METHOD PROTECTED M_ProcessFCR : BOOL
(**************************************************************************************
 * 	Application		:	BoxControl Framework
 *	Revision		:	$Revision: 404529 $
 *	Revision date	:	$Date: 2018-04-23 08:21:38 +0200 (Mo., 23 Apr 2018) $
 *	Last changed by	:	$Author: b7bolm $
 *	URL				:	$URL: http://almscdc.swisslog.com/repo/SWPD/Development/BoxControlFramework/20_Release/trunk/01_Software/BCF/BCF/JumpStart/20_Product/10_App/11_Com/10_Lib/10_Conv/12_MFCS/11_SIS/FB_SIS_MsgManager_6_1.TcPOU $
 *
 *	Purpose			:	Send FCR
 *
 * ------------------------------------------------------------------------------------
 *	Copyright Swisslog [IP AG], Switzerland. All rights reserved.
 * 
 * ------------------------------------------------------------------------------------
 *	
 * 	Revision History: 
 *
 * 	VERSION			DATE			INITIALS			DESCRIPTION
 *	0.1				01.01.2001		swl					Example
 *
 **************************************************************************************)
VAR_INPUT
 	meChannelSrc		: E_MFCS_Channel; // Source communicaton channel
	mpFCR				: POINTER TO ST_ITC_FCR; // Pointer to FCR
END_VAR
(**************************************************************************************************************
 	Check if a telegram needs to be send
***************************************************************************************************************)
// If settings allow sending a FCR 	
IF  Settings.Telegrams.SendFCR THEN
	// If the source of the request is this channel or is undefined
	IF meChannelSrc = Settings.MFCS_Channel OR
		meChannelSrc = E_MFCS_Channel.BEGIN_CHANNEL THEN
		;//Proceed
	ELSE // Source is a different MFCS Connection
		// Dont send a telegram		
		RETURN;
	END_IF	
ELSE
	// Dont send a telegram		
	RETURN;
END_IF

(**************************************************************************************************************
 	ITC - Map generic data to type
***************************************************************************************************************)
MEMCPY(destAddr := ADR(FCR_ITC), srcAddr := mpFCR, n := SIZEOF(FCR_ITC));

(**************************************************************************************************************
 	Formatting data
***************************************************************************************************************)

// Fill position
FCR.Position	:= 	F_StuffString(
						InputString 	:= FCR_ITC.Position, 
						StringLength	:= SIS_6_1.POSITION_STRINGLENGTH, 
						StuffCharacter 	:= '0',
						LeftAligned		:= FALSE);

// Fill code
FCR.Code	:= F_StuffString(
				InputString 	:= INT_TO_STRING(FCR_ITC.Code), 
				StringLength	:= SIS_6_1.CONTROLCODE_STRINGLENGTH, 
				StuffCharacter 	:= '0',
				LeftAligned		:= FALSE);

// Fill variable
FCR.Variable 	:= F_StuffString(
					InputString 	:= DINT_TO_STRING(FCR_ITC.Variable), 
					StringLength	:= SIS_6_1.CONTROLVARIABLE_STRINGLENGTH, 
					StuffCharacter 	:= '0',
					LeftAligned		:= FALSE);

// Fill errorcode
FCR.ReturnCode 	:= F_StuffString(
					InputString 	:= INT_TO_STRING(FCR_ITC.ReturnCode), 
					StringLength	:= SIS_6_1.ERRORCODE_STRINGLENGTH, 
					StuffCharacter 	:= '0',
					LeftAligned		:= FALSE);


(**************************************************************************************************************
 	Build string and add to Base Driver
***************************************************************************************************************)
MEMSET(destAddr := ADR(SendTelegram), 0, SIZEOF(SendTelegram));
WritePointer := 0;

F_AssembleByteStream(
	pSrc:= ADR('FCR'), 
	SrcLen:= 3, 
	pDest:= ADR(SendTelegram), 
	DestLen:= SIZEOF(SendTelegram), 
	WritePointer:= WritePointer);

F_AssembleByteStream(
	pSrc:= ADR(FCR.Position), 
	SrcLen:= INT_TO_UDINT(LEN(FCR.Position)), 
	pDest:= ADR(SendTelegram), 
	DestLen:= SIZEOF(SendTelegram), 
	WritePointer:= WritePointer);	
	
F_AssembleByteStream(
	pSrc:= ADR(FCR.Code), 
	SrcLen:= INT_TO_UDINT(LEN(FCR.Code)), 
	pDest:= ADR(SendTelegram), 
	DestLen:= SIZEOF(SendTelegram), 
	WritePointer:= WritePointer);	
	
F_AssembleByteStream(
	pSrc:= ADR(FCR.Variable), 
	SrcLen:= INT_TO_UDINT(LEN(FCR.Variable)), 
	pDest:= ADR(SendTelegram), 
	DestLen:= SIZEOF(SendTelegram), 
	WritePointer:= WritePointer);	
	
F_AssembleByteStream(
	pSrc:= ADR(FCR.ReturnCode), 
	SrcLen:= INT_TO_UDINT(LEN(FCR.ReturnCode)), 
	pDest:= ADR(SendTelegram), 
	DestLen:= SIZEOF(SendTelegram), 
	WritePointer:= WritePointer);	

// Add to buffer of Base Driver
M_ProcessFCR := fbBaseDriver.M_SendAppData(
					mpSendData := ADR(SendTelegram),
					mSendDataLen := WritePointer);
					
// Forward to mirror channel
M_MirrorData(Data := ADR(SendTelegram), DataLen := WritePointer);
END_METHOD

METHOD PROTECTED M_ProcessFSR : BOOL
(**************************************************************************************
 * 	Application		:	BoxControl Framework
 *	Revision		:	$Revision: 404529 $
 *	Revision date	:	$Date: 2018-04-23 08:21:38 +0200 (Mo., 23 Apr 2018) $
 *	Last changed by	:	$Author: b7bolm $
 *	URL				:	$URL: http://almscdc.swisslog.com/repo/SWPD/Development/BoxControlFramework/20_Release/trunk/01_Software/BCF/BCF/JumpStart/20_Product/10_App/11_Com/10_Lib/10_Conv/12_MFCS/11_SIS/FB_SIS_MsgManager_6_1.TcPOU $
 *
 *	Purpose			:	Send FSR
 *
 * ------------------------------------------------------------------------------------
 *	Copyright Swisslog [IP AG], Switzerland. All rights reserved.
 * 
 * ------------------------------------------------------------------------------------
 *	
 * 	Revision History: 
 *
 * 	VERSION			DATE			INITIALS			DESCRIPTION
 *	0.1				01.01.2001		swl					Example
 *
 **************************************************************************************)
VAR_INPUT
 	meChannelSrc		: E_MFCS_Channel; // Source communicaton channel
	mpFSR				: POINTER TO ST_ITC_FSR; // Pointer to FSR
END_VAR
(**************************************************************************************************************
 	Check if a telegram needs to be send
***************************************************************************************************************)
// If settings allow sending a FSR 	
IF  Settings.Telegrams.SendFSR THEN
	// If the source of the request is this channel or is undefined
	IF meChannelSrc = Settings.MFCS_Channel OR
		meChannelSrc = E_MFCS_Channel.BEGIN_CHANNEL THEN
		;//Proceed
	ELSE // Source is a different MFCS Connection
		// Dont send a telegram		
		RETURN;
	END_IF	
ELSE
	// Dont send a telegram		
	RETURN;
END_IF

(**************************************************************************************************************
 	ITC - Map generic data to type
***************************************************************************************************************)
MEMCPY(destAddr := ADR(FSR_ITC), srcAddr := mpFSR, n := SIZEOF(FSR_ITC));

(**************************************************************************************************************
 	Formatting data
***************************************************************************************************************)
// Set position
FSR.Position := F_StuffString(
					InputString 	:= FSR_ITC.Position, 
					StringLength	:= SIS_6_1.POSITION_STRINGLENGTH, 
					StuffCharacter 	:= '0',
					LeftAligned		:= FALSE);
					
// Set previous function no
FSR.PrevFunctionNo := F_StuffString(
						InputString 	:= FSR_ITC.PrevFunctionNo, 
						StringLength	:= SIS_6_1.POSITION_STRINGLENGTH, 
						StuffCharacter 	:= '0',
						LeftAligned		:= FALSE);
						
// Set next function no
FSR.NextFunctionNo := F_StuffString(
						InputString 	:= FSR_ITC.NextFunctionNo, 
						StringLength	:= SIS_6_1.POSITION_STRINGLENGTH, 
						StuffCharacter 	:= '0',
						LeftAligned		:= FALSE);
						
// Set state
FSR.State := INT_TO_STRING(FSR_ITC.eState);

// Set enabled
FSR.Enabled := INT_TO_STRING(BOOL_TO_INT(FSR_ITC.Enabled));

//modifications needed BCFD-10111FSR data incorrect (M_ProcessFSR)
// Set transport state
FSR.TransportState := F_StuffString(
						InputString 	:= INT_TO_STRING(TO_INT(FSR_ITC.TransportState)), 
						StringLength	:= SIS_6_1.FSR_STATES_STRINGLENGTH, 
						StuffCharacter 	:= '0',
						LeftAligned		:= FALSE);

// Set takeover state	
FSR.TakeOverState := F_StuffString(
						InputString 	:= INT_TO_STRING(TO_INT(FSR_ITC.TakeOverState)), 
						StringLength	:= SIS_6_1.FSR_STATES_STRINGLENGTH, 
						StuffCharacter 	:= '0',
						LeftAligned		:= FALSE);

// Set handover state
FSR.HandOverState := F_StuffString(
						InputString 	:= INT_TO_STRING(TO_INT(FSR_ITC.HandOverState)), 
						StringLength	:= SIS_6_1.FSR_STATES_STRINGLENGTH, 
						StuffCharacter 	:= '0',
						LeftAligned		:= FALSE);

// Set TU-ID
FSR.TU_ID := F_StuffString(
				InputString 	:= FSR_ITC.TU_ID, 
				StringLength	:= SIS_6_1.TU_ID_STRINGLENGTH, 
				StuffCharacter 	:= ' ',
				LeftAligned		:= FALSE);

// Set TU-Type	
FSR.TU_Type := F_StuffString(
				InputString 	:= INT_TO_STRING(FSR_ITC.TU_Type), 
				StringLength	:= SIS_6_1.TU_TYPE_STRINGLENGTH, 
				StuffCharacter 	:= '0',
				LeftAligned		:= FALSE);
				
// Set Assignment ID	
FSR.AssignmentID := F_StuffString(
						InputString 	:= UDINT_TO_STRING(FSR_ITC.AssignmentID), 
						StringLength	:= SIS_6_1.ASSIGNMENT_ID_STRINGLENGTH, 
						StuffCharacter 	:= '0',
						LeftAligned		:= FALSE);

// Set load information	
FSR.LoadInformation  := INT_TO_STRING(FSR_ITC.LoadInformation);

// Set destination
FSR.Destination  := F_StuffString(
						InputString 	:= FSR_ITC.Destination, 
						StringLength	:= SIS_6_1.POSITION_STRINGLENGTH, 
						StuffCharacter 	:= '0',
						LeftAligned		:= FALSE);
						
// Set error state
FSR.ErrorState := INT_TO_STRING(FSR_ITC.eErrorState);

// Set error code				
FSR.ErrorCode := F_StuffString(
					InputString 	:= INT_TO_STRING(FSR_ITC.eErrorCode), 
					StringLength	:= SIS_6_1.ERRORCODE_STRINGLENGTH, 
					StuffCharacter 	:= '0',
					LeftAligned		:= FALSE);
					
// Set error type		
FSR.ErrorType  := INT_TO_STRING(FSR_ITC.eErrorType);

// Set error information	
FSR.ErrorInformation  := F_StuffString(
							InputString 	:= FSR_ITC.ErrorInformation, 
							StringLength	:= SIS_6_1.ERRORINFORMATION_STRINGLENGTH, 
							StuffCharacter 	:= ' ',
							LeftAligned		:= TRUE);
// Set variable		
FSR.Variable := F_StuffString(
					InputString 	:= DINT_TO_STRING(FSR_ITC.Variable), 
					StringLength	:= SIS_6_1.FSR_VARIABLE_STRINGLENGTH, 
					StuffCharacter 	:= '0',
					LeftAligned		:= FALSE);

// Get Error Code 
FSR.ReturnCode := F_StuffString(
					InputString 	:= INT_TO_STRING(FSR_ITC.eReturnCode), 
					StringLength	:= SIS_6_1.ERRORCODE_STRINGLENGTH, 
					StuffCharacter 	:= '0',
					LeftAligned		:= FALSE);
					
(**************************************************************************************************************
 	Build string and add to Base Driver
***************************************************************************************************************)
MEMSET(destAddr := ADR(SendTelegram), 0, SIZEOF(SendTelegram));
WritePointer := 0;

F_AssembleByteStream(
	pSrc:= ADR('FSR'), 
	SrcLen:= 3, 
	pDest:= ADR(SendTelegram), 
	DestLen:= SIZEOF(SendTelegram), 
	WritePointer:= WritePointer);

F_AssembleByteStream(
	pSrc:= ADR(FSR.Position), 
	SrcLen:= INT_TO_UDINT(LEN(FSR.Position)), 
	pDest:= ADR(SendTelegram), 
	DestLen:= SIZEOF(SendTelegram), 
	WritePointer:= WritePointer);	

F_AssembleByteStream(
	pSrc:= ADR(FSR.PrevFunctionNo), 
	SrcLen:= INT_TO_UDINT(LEN(FSR.PrevFunctionNo)), 
	pDest:= ADR(SendTelegram), 
	DestLen:= SIZEOF(SendTelegram), 
	WritePointer:= WritePointer);	

F_AssembleByteStream(
	pSrc:= ADR(FSR.NextFunctionNo), 
	SrcLen:= INT_TO_UDINT(LEN(FSR.NextFunctionNo)), 
	pDest:= ADR(SendTelegram), 
	DestLen:= SIZEOF(SendTelegram), 
	WritePointer:= WritePointer);	
	
F_AssembleByteStream(
	pSrc:= ADR(FSR.State), 
	SrcLen:= INT_TO_UDINT(LEN(FSR.State)), 
	pDest:= ADR(SendTelegram), 
	DestLen:= SIZEOF(SendTelegram), 
	WritePointer:= WritePointer);	
	
F_AssembleByteStream(
	pSrc:= ADR(FSR.Enabled), 
	SrcLen:= INT_TO_UDINT(LEN(FSR.Enabled)), 
	pDest:= ADR(SendTelegram), 
	DestLen:= SIZEOF(SendTelegram), 
	WritePointer:= WritePointer);	
	
F_AssembleByteStream(
	pSrc:= ADR(FSR.TransportState), 
	SrcLen:= INT_TO_UDINT(LEN(FSR.TransportState)), 
	pDest:= ADR(SendTelegram), 
	DestLen:= SIZEOF(SendTelegram), 
	WritePointer:= WritePointer);	
	
F_AssembleByteStream(
	pSrc:= ADR(FSR.TakeOverState), 
	SrcLen:= INT_TO_UDINT(LEN(FSR.TakeOverState)), 
	pDest:= ADR(SendTelegram), 
	DestLen:= SIZEOF(SendTelegram), 
	WritePointer:= WritePointer);	
	
F_AssembleByteStream(
	pSrc:= ADR(FSR.HandOverState), 
	SrcLen:= INT_TO_UDINT(LEN(FSR.HandOverState)), 
	pDest:= ADR(SendTelegram), 
	DestLen:= SIZEOF(SendTelegram), 
	WritePointer:= WritePointer);	

F_AssembleByteStream(
	pSrc:= ADR(FSR.TU_ID), 
	SrcLen:= INT_TO_UDINT(LEN(FSR.TU_ID)), 
	pDest:= ADR(SendTelegram), 
	DestLen:= SIZEOF(SendTelegram), 
	WritePointer:= WritePointer);	
	
F_AssembleByteStream(
	pSrc:= ADR(FSR.TU_Type), 
	SrcLen:= INT_TO_UDINT(LEN(FSR.TU_Type)), 
	pDest:= ADR(SendTelegram), 
	DestLen:= SIZEOF(SendTelegram), 
	WritePointer:= WritePointer);	

F_AssembleByteStream(
	pSrc:= ADR(FSR.AssignmentID), 
	SrcLen:= INT_TO_UDINT(LEN(FSR.AssignmentID)), 
	pDest:= ADR(SendTelegram), 
	DestLen:= SIZEOF(SendTelegram), 
	WritePointer:= WritePointer);	

F_AssembleByteStream(
	pSrc:= ADR(FSR.LoadInformation), 
	SrcLen:= INT_TO_UDINT(LEN(FSR.LoadInformation)), 
	pDest:= ADR(SendTelegram), 
	DestLen:= SIZEOF(SendTelegram), 
	WritePointer:= WritePointer);	
	
F_AssembleByteStream(
	pSrc:= ADR(FSR.Destination), 
	SrcLen:= INT_TO_UDINT(LEN(FSR.Destination)), 
	pDest:= ADR(SendTelegram), 
	DestLen:= SIZEOF(SendTelegram), 
	WritePointer:= WritePointer);	

F_AssembleByteStream(
	pSrc:= ADR(FSR.ErrorState), 
	SrcLen:= INT_TO_UDINT(LEN(FSR.ErrorState)), 
	pDest:= ADR(SendTelegram), 
	DestLen:= SIZEOF(SendTelegram), 
	WritePointer:= WritePointer);	
		
F_AssembleByteStream(
	pSrc:= ADR(FSR.ErrorCode), 
	SrcLen:= INT_TO_UDINT(LEN(FSR.ErrorCode)), 
	pDest:= ADR(SendTelegram), 
	DestLen:= SIZEOF(SendTelegram), 
	WritePointer:= WritePointer);	
	
F_AssembleByteStream(
	pSrc:= ADR(FSR.ErrorType), 
	SrcLen:= INT_TO_UDINT(LEN(FSR.ErrorType)), 
	pDest:= ADR(SendTelegram), 
	DestLen:= SIZEOF(SendTelegram), 
	WritePointer:= WritePointer);	
	
F_AssembleByteStream(
	pSrc:= ADR(FSR.ErrorInformation), 
	SrcLen:= INT_TO_UDINT(LEN(FSR.ErrorInformation)), 
	pDest:= ADR(SendTelegram), 
	DestLen:= SIZEOF(SendTelegram), 
	WritePointer:= WritePointer);	
	
F_AssembleByteStream(
	pSrc:= ADR(FSR.Variable), 
	SrcLen:= INT_TO_UDINT(LEN(FSR.Variable)), 
	pDest:= ADR(SendTelegram), 
	DestLen:= SIZEOF(SendTelegram), 
	WritePointer:= WritePointer);	
	
F_AssembleByteStream(
	pSrc:= ADR(FSR.ReturnCode), 
	SrcLen:= INT_TO_UDINT(LEN(FSR.ReturnCode)), 
	pDest:= ADR(SendTelegram), 
	DestLen:= SIZEOF(SendTelegram), 
	WritePointer:= WritePointer);	
	

// Add to buffer of Base Driver
M_ProcessFSR := fbBaseDriver.M_SendAppData(
					mpSendData := ADR(SendTelegram),
					mSendDataLen := WritePointer);

// Forward to mirror channel
M_MirrorData(Data := ADR(SendTelegram), DataLen := WritePointer);
END_METHOD

METHOD PROTECTED M_ProcessGCR : BOOL
(**************************************************************************************
 * 	Application		:	BoxControl Framework
 *	Revision		:	$Revision: 404529 $
 *	Revision date	:	$Date: 2018-04-23 08:21:38 +0200 (Mo., 23 Apr 2018) $
 *	Last changed by	:	$Author: b7bolm $
 *	URL				:	$URL: http://almscdc.swisslog.com/repo/SWPD/Development/BoxControlFramework/20_Release/trunk/01_Software/BCF/BCF/JumpStart/20_Product/10_App/11_Com/10_Lib/10_Conv/12_MFCS/11_SIS/FB_SIS_MsgManager_6_1.TcPOU $
 *
 *	Purpose			:	Send GCR
 *
 * ------------------------------------------------------------------------------------
 *	Copyright Swisslog [IP AG], Switzerland. All rights reserved.
 * 
 * ------------------------------------------------------------------------------------
 *	
 * 	Revision History: 
 *
 * 	VERSION			DATE			INITIALS			DESCRIPTION
 *	0.1				01.01.2001		swl					Example
 *
 **************************************************************************************)
VAR_INPUT
 	meChannelSrc		: E_MFCS_Channel; // Source communicaton channel
	mpGCR				: POINTER TO ST_ITC_GCR; // Pointer to GCR
END_VAR
(**************************************************************************************************************
 	Check if a telegram needs to be send
***************************************************************************************************************)
// If settings allow sending a GCR 	
IF  Settings.Telegrams.SendGCR THEN
	// If the source of the request is this channel or is undefined
	IF meChannelSrc = Settings.MFCS_Channel OR
		meChannelSrc = E_MFCS_Channel.BEGIN_CHANNEL THEN
		;//Proceed
	ELSE // Source is a different MFCS Connection
		// Dont send a telegram		
		RETURN;
	END_IF	
ELSE
	// Dont send a telegram		
	RETURN;
END_IF

(**************************************************************************************************************
 	ITC - Map generic data to type
***************************************************************************************************************)
MEMCPY(destAddr := ADR(GCR_ITC), srcAddr := mpGCR, n := SIZEOF(GCR_ITC));

(**************************************************************************************************************
 	Formatting data
***************************************************************************************************************)
// Get SIS-Number 
GCR.GroupName := F_StuffString(
					InputString 	:= GCR_ITC.GroupName, 
					StringLength	:= SIS_6_1.POSITION_STRINGLENGTH, 
					StuffCharacter 	:= '0',
					LeftAligned		:= FALSE);

// Get Code 
GCR.Code := F_StuffString(
				InputString 	:= INT_TO_STRING(GCR_ITC.Code), 
				StringLength	:= SIS_6_1.CONTROLCODE_STRINGLENGTH, 
				StuffCharacter 	:= '0',
				LeftAligned		:= FALSE);

// Get Variable 
GCR.Variable := F_StuffString(
					InputString 	:= DINT_TO_STRING(GCR_ITC.Variable), 
					StringLength	:= SIS_6_1.CONTROLVARIABLE_STRINGLENGTH, 
					StuffCharacter 	:= '0',
					LeftAligned		:= FALSE);

// Get ErrorCode 
GCR.ReturnCode := F_StuffString(
					InputString 	:= INT_TO_STRING(GCR_ITC.ReturnCode), 
					StringLength	:= SIS_6_1.ERRORCODE_STRINGLENGTH, 
					StuffCharacter 	:= '0',
					LeftAligned		:= FALSE);

(**************************************************************************************************************
 	Build string and add to Base Driver
***************************************************************************************************************)
MEMSET(destAddr := ADR(SendTelegram), 0, SIZEOF(SendTelegram));
WritePointer := 0;

F_AssembleByteStream(
	pSrc:= ADR('GCR'), 
	SrcLen:= 3, 
	pDest:= ADR(SendTelegram), 
	DestLen:= SIZEOF(SendTelegram), 
	WritePointer:= WritePointer);

F_AssembleByteStream(
	pSrc:= ADR(GCR.GroupName), 
	SrcLen:= INT_TO_UDINT(LEN(GCR.GroupName)), 
	pDest:= ADR(SendTelegram), 
	DestLen:= SIZEOF(SendTelegram), 
	WritePointer:= WritePointer);	

F_AssembleByteStream(
	pSrc:= ADR(GCR.Code), 
	SrcLen:= INT_TO_UDINT(LEN(GCR.Code)), 
	pDest:= ADR(SendTelegram), 
	DestLen:= SIZEOF(SendTelegram), 
	WritePointer:= WritePointer);	

F_AssembleByteStream(
	pSrc:= ADR(GCR.Variable), 
	SrcLen:= INT_TO_UDINT(LEN(GCR.Variable)), 
	pDest:= ADR(SendTelegram), 
	DestLen:= SIZEOF(SendTelegram), 
	WritePointer:= WritePointer);	

F_AssembleByteStream(
	pSrc:= ADR(GCR.ReturnCode), 
	SrcLen:= INT_TO_UDINT(LEN(GCR.ReturnCode)), 
	pDest:= ADR(SendTelegram), 
	DestLen:= SIZEOF(SendTelegram), 
	WritePointer:= WritePointer);	

// Add to buffer of Base Driver
M_ProcessGCR := fbBaseDriver.M_SendAppData(
					mpSendData := ADR(SendTelegram),
					mSendDataLen := WritePointer);

// Forward to mirror channel
M_MirrorData(Data := ADR(SendTelegram), DataLen := WritePointer);
END_METHOD

METHOD PROTECTED M_ProcessGDR : BOOL
(**************************************************************************************
 * 	Application		:	BoxControl Framework
 *	Revision		:	$Revision: 404529 $
 *	Revision date	:	$Date: 2018-04-23 08:21:38 +0200 (Mo., 23 Apr 2018) $
 *	Last changed by	:	$Author: b7bolm $
 *	URL				:	$URL: http://almscdc.swisslog.com/repo/SWPD/Development/BoxControlFramework/20_Release/trunk/01_Software/BCF/BCF/JumpStart/20_Product/10_App/11_Com/10_Lib/10_Conv/12_MFCS/11_SIS/FB_SIS_MsgManager_6_1.TcPOU $
 *
 *	Purpose			:	Send GDR
 *
 * ------------------------------------------------------------------------------------
 *	Copyright Swisslog [IP AG], Switzerland. All rights reserved.
 * 
 * ------------------------------------------------------------------------------------
 *	
 * 	Revision History: 
 *
 * 	VERSION			DATE			INITIALS			DESCRIPTION
 *	0.1				01.01.2001		swl					Example
 *
 **************************************************************************************)
VAR_INPUT
 	meChannelSrc		: E_MFCS_Channel; // Source communicaton channel
	mpGDR				: POINTER TO ST_ITC_GDR; // Pointer to GDR
END_VAR
(**************************************************************************************************************
 	Check if a telegram needs to be send
***************************************************************************************************************)
// If settings allow sending a GDR 	
IF  Settings.Telegrams.SendGDR THEN
	// If the source of the request is this channel or is undefined
	IF meChannelSrc = Settings.MFCS_Channel OR
		meChannelSrc = E_MFCS_Channel.BEGIN_CHANNEL THEN
		;//Proceed
	ELSE // Source is a different MFCS Connection
		// Dont send a telegram		
		RETURN;
	END_IF	
ELSE
	// Dont send a telegram		
	RETURN;
END_IF

(**************************************************************************************************************
 	ITC - Map generic data to type
***************************************************************************************************************)
MEMCPY(destAddr := ADR(GDR_ITC), srcAddr := mpGDR, n := SIZEOF(GDR_ITC));
MEMSET(destAddr := ADR(GDR), 0, SIZEOF(GDR));
(**************************************************************************************************************
 	Formatting data
***************************************************************************************************************)
// Get SIS-Number 
GDR.Position := F_StuffString(
					InputString 	:= GDR_ITC.Position, 
					StringLength	:= SIS_6_1.POSITION_STRINGLENGTH, 
					StuffCharacter 	:= '0',
					LeftAligned := FALSE);
// Get Variable 
GDR.Variable := F_StuffString(
				InputString 	:= GDR_ITC.Variable, 
				StringLength	:= SIS_6_1.GATHERED_DATA_VARIABLE, 
				StuffCharacter 	:= ' ',
				LeftAligned		:= FALSE);
//Number of Sets
GDR.NumberOfSets := 	F_StuffString(
										InputString 	:=INT_TO_STRING(GDR_ITC.NumberOfSets), 
										StringLength	:= SIS_6_1.DATA_ACQUISITION_NUMBEROFSETS, 
										StuffCharacter 	:= '0',
										LeftAligned		:= FALSE);
//Build Data Set String
FOR Idx:= 0 TO GDR_ITC.NumberOfSets-1 DO 
	GDR.DataSet[Idx]  := CONCAT(GDR.DataSet[Idx],F_StuffString(InputString := GDR_ITC.DataSet[Idx].Value, StringLength:= Conveyor.GATHERED_DATA_VALUE,StuffCharacter := '0', LeftAligned := FALSE));
	GDR.DataSet[Idx]  := CONCAT(GDR.DataSet[Idx],GDR_ITC.DataSet[Idx].TimeStamp);
	GDR.DataSet[Idx]  := CONCAT(GDR.DataSet[Idx],F_StuffString(InputString 	:= INT_TO_STRING(GDR_ITC.DataSet[Idx].Sequence), StringLength:= SIS_6_1.GATHERED_DATA_SEQUENCE,StuffCharacter := '0', LeftAligned := FALSE));
END_FOR;

// Get Error Code 
GDR.ReturnCode := F_StuffString(
				InputString 	:= INT_TO_STRING(GDR_ITC.eReturnCode), 
				StringLength	:= SIS_6_1.ERRORCODE_STRINGLENGTH, 
				StuffCharacter 	:= '0',
				LeftAligned 	:= FALSE);
				
(**************************************************************************************************************
 	Build string and add to Base Driver
***************************************************************************************************************)
MEMSET(destAddr := ADR(SendTelegram), 0, SIZEOF(SendTelegram));
WritePointer := 0;

F_AssembleByteStream(
	pSrc:= ADR('GDR'), 
	SrcLen:= 3, 
	pDest:= ADR(SendTelegram), 
	DestLen:= SIZEOF(SendTelegram), 
	WritePointer:= WritePointer);
	
F_AssembleByteStream(
	pSrc:= ADR(GDR.Position), 
	SrcLen:= INT_TO_UDINT(LEN(GDR.Position)), 
	pDest:= ADR(SendTelegram), 
	DestLen:= SIZEOF(SendTelegram), 
	WritePointer:= WritePointer);

F_AssembleByteStream(
	pSrc:= ADR(GDR.Variable), 
	SrcLen:= INT_TO_UDINT(LEN(GDR.Variable)), 
	pDest:= ADR(SendTelegram), 
	DestLen:= SIZEOF(SendTelegram), 
	WritePointer:= WritePointer);

F_AssembleByteStream(
	pSrc:= ADR(GDR.NumberOfSets), 
	SrcLen:= INT_TO_UDINT(LEN(GDR.NumberOfSets)), 
	pDest:= ADR(SendTelegram), 
	DestLen:= SIZEOF(SendTelegram), 
	WritePointer:= WritePointer);

FOR Idx:= 0
 TO GDR_ITC.NumberOfSets DO
	F_AssembleByteStream(
						pSrc		:= ADR(GDR.DataSet[Idx]), 
						SrcLen		:= INT_TO_UDINT(LEN(GDR.DataSet[Idx])), 
						pDest		:= ADR(SendTelegram),
						DestLen		:= SIZEOF(SendTelegram), 
						WritePointer:= WritePointer);
						
END_FOR

	
	
	
F_AssembleByteStream(
	pSrc:= ADR(GDR.ReturnCode), 
	SrcLen:= INT_TO_UDINT(LEN(GDR.ReturnCode)), 
	pDest:= ADR(SendTelegram), 
	DestLen:= SIZEOF(SendTelegram), 
	WritePointer:= WritePointer);

// Add to buffer of Base Driver
M_ProcessGDR := fbBaseDriver.M_SendAppData(
					mpSendData := ADR(SendTelegram),
					mSendDataLen := WritePointer);

// Forward to mirror channel
M_MirrorData(Data := ADR(SendTelegram), DataLen := WritePointer);
END_METHOD

METHOD PROTECTED M_ProcessGSR : BOOL
(**************************************************************************************
 * 	Application		:	BoxControl Framework
 *	Revision		:	$Revision: 404529 $
 *	Revision date	:	$Date: 2018-04-23 08:21:38 +0200 (Mo., 23 Apr 2018) $
 *	Last changed by	:	$Author: b7bolm $
 *	URL				:	$URL: http://almscdc.swisslog.com/repo/SWPD/Development/BoxControlFramework/20_Release/trunk/01_Software/BCF/BCF/JumpStart/20_Product/10_App/11_Com/10_Lib/10_Conv/12_MFCS/11_SIS/FB_SIS_MsgManager_6_1.TcPOU $
 *
 *	Purpose			:	Send GSR
 *
 * ------------------------------------------------------------------------------------
 *	Copyright Swisslog [IP AG], Switzerland. All rights reserved.
 * 
 * ------------------------------------------------------------------------------------
 *	
 * 	Revision History: 
 *
 * 	VERSION			DATE			INITIALS			DESCRIPTION
 *	0.1				01.01.2001		swl					Example
 *
 **************************************************************************************)
VAR_INPUT
 	meChannelSrc		: E_MFCS_Channel; // Source communicaton channel
	mpGSR				: POINTER TO ST_ITC_GSR; // Pointer to GSR
END_VAR
(**************************************************************************************************************
 	Check if a telegram needs to be send
***************************************************************************************************************)
// If settings allow sending a GSR 	
IF  Settings.Telegrams.SendGSR THEN
	// If the source of the request is this channel or is undefined
	IF meChannelSrc = Settings.MFCS_Channel OR
		meChannelSrc = E_MFCS_Channel.BEGIN_CHANNEL THEN
		;//Proceed
	ELSE // Source is a different MFCS Connection
		// Dont send a telegram		
		RETURN;
	END_IF	
ELSE
	// Dont send a telegram		
	RETURN;
END_IF

(**************************************************************************************************************
 	ITC - Map generic data to type
***************************************************************************************************************)
MEMCPY(destAddr := ADR(GSR_ITC), srcAddr := mpGSR, n := SIZEOF(GSR_ITC));

(**************************************************************************************************************
 	Formatting data
***************************************************************************************************************)
// Get SIS-Number 
GSR.GroupName := F_StuffString(
					InputString 	:= GSR_ITC.GroupName, 
					StringLength	:= SIS_6_1.POSITION_STRINGLENGTH, 
					StuffCharacter 	:= '0',
					LeftAligned		:= FALSE);

// Get Mode 
GSR.Mode := INT_TO_STRING(GSR_ITC.eMode);

// Get State 
GSR.State := INT_TO_STRING(GSR_ITC.eState);

// Get ErrorState 
GSR.ErrorState := INT_TO_STRING(GSR_ITC.eErrorState);

// Get ErrorCode 
GSR.ErrorCode := F_StuffString(
					InputString 	:= INT_TO_STRING(GSR_ITC.eErrorCode), 
					StringLength	:= SIS_6_1.ERRORCODE_STRINGLENGTH, 
					StuffCharacter 	:= '0',
					LeftAligned		:= FALSE);

// Get ErrorType 
GSR.ErrorType := INT_TO_STRING(GSR_ITC.eErrorType);

// Get ErrorInformation 
GSR.ErrorInformation := F_StuffString(
							InputString 	:= GSR_ITC.ErrorInformation, 
							StringLength	:= SIS_6_1.ERRORINFORMATION_STRINGLENGTH, 
							StuffCharacter 	:= ' ',
							LeftAligned		:= TRUE);

// Get Variable 
GSR.Variable := F_StuffString(
					InputString 	:= DINT_TO_STRING(GSR_ITC.Variable), 
					StringLength	:= SIS_6_1.CONTROLVARIABLE_STRINGLENGTH, 
					StuffCharacter 	:= '0',
					LeftAligned		:= FALSE);
					
// Get Error Code 
GSR.ReturnCode := F_StuffString(
					InputString 	:= INT_TO_STRING(GSR_ITC.eReturnCode), 
					StringLength	:= SIS_6_1.ERRORCODE_STRINGLENGTH, 
					StuffCharacter 	:= '0',
					LeftAligned		:= FALSE);

(**************************************************************************************************************
 	Build string and add to Base Driver
***************************************************************************************************************)
MEMSET(destAddr := ADR(SendTelegram), 0, SIZEOF(SendTelegram));
WritePointer := 0;

F_AssembleByteStream(
	pSrc:= ADR('GSR'), 
	SrcLen:= 3, 
	pDest:= ADR(SendTelegram), 
	DestLen:= SIZEOF(SendTelegram), 
	WritePointer:= WritePointer);

F_AssembleByteStream(
	pSrc:= ADR(GSR.GroupName), 
	SrcLen:= INT_TO_UDINT(LEN(GSR.GroupName)), 
	pDest:= ADR(SendTelegram), 
	DestLen:= SIZEOF(SendTelegram), 
	WritePointer:= WritePointer);	
	
F_AssembleByteStream(
	pSrc:= ADR(GSR.Mode), 
	SrcLen:= INT_TO_UDINT(LEN(GSR.Mode)), 
	pDest:= ADR(SendTelegram), 
	DestLen:= SIZEOF(SendTelegram), 
	WritePointer:= WritePointer);	
	
F_AssembleByteStream(
	pSrc:= ADR(GSR.State), 
	SrcLen:= INT_TO_UDINT(LEN(GSR.State)), 
	pDest:= ADR(SendTelegram), 
	DestLen:= SIZEOF(SendTelegram), 
	WritePointer:= WritePointer);	

F_AssembleByteStream(
	pSrc:= ADR(GSR.ErrorState), 
	SrcLen:= INT_TO_UDINT(LEN(GSR.ErrorState)), 
	pDest:= ADR(SendTelegram), 
	DestLen:= SIZEOF(SendTelegram), 
	WritePointer:= WritePointer);	

F_AssembleByteStream(
	pSrc:= ADR(GSR.ErrorCode), 
	SrcLen:= INT_TO_UDINT(LEN(GSR.ErrorCode)), 
	pDest:= ADR(SendTelegram), 
	DestLen:= SIZEOF(SendTelegram), 
	WritePointer:= WritePointer);	
	
F_AssembleByteStream(
	pSrc:= ADR(GSR.ErrorType), 
	SrcLen:= INT_TO_UDINT(LEN(GSR.ErrorType)), 
	pDest:= ADR(SendTelegram), 
	DestLen:= SIZEOF(SendTelegram), 
	WritePointer:= WritePointer);	
	
F_AssembleByteStream(
	pSrc:= ADR(GSR.ErrorInformation), 
	SrcLen:= INT_TO_UDINT(LEN(GSR.ErrorInformation)), 
	pDest:= ADR(SendTelegram), 
	DestLen:= SIZEOF(SendTelegram), 
	WritePointer:= WritePointer);	

F_AssembleByteStream(
	pSrc:= ADR(GSR.Variable), 
	SrcLen:= INT_TO_UDINT(LEN(GSR.Variable)), 
	pDest:= ADR(SendTelegram), 
	DestLen:= SIZEOF(SendTelegram), 
	WritePointer:= WritePointer);	
	
F_AssembleByteStream(
	pSrc:= ADR(GSR.ReturnCode), 
	SrcLen:= INT_TO_UDINT(LEN(GSR.ReturnCode)), 
	pDest:= ADR(SendTelegram), 
	DestLen:= SIZEOF(SendTelegram), 
	WritePointer:= WritePointer);	


// Add to buffer of Base Driver
M_ProcessGSR := fbBaseDriver.M_SendAppData(
					mpSendData := ADR(SendTelegram),
					mSendDataLen := WritePointer);

// Forward to mirror channel
M_MirrorData(Data := ADR(SendTelegram), DataLen := WritePointer);
END_METHOD

METHOD PROTECTED M_ProcessGVR : BOOL
(**************************************************************************************
 * 	Application		:	BoxControl Framework
 *	Revision		:	$Revision: 404529 $
 *	Revision date	:	$Date: 2018-04-23 08:21:38 +0200 (Mo., 23 Apr 2018) $
 *	Last changed by	:	$Author: b7bolm $
 *	URL				:	$URL: http://almscdc.swisslog.com/repo/SWPD/Development/BoxControlFramework/20_Release/trunk/01_Software/BCF/BCF/JumpStart/20_Product/10_App/11_Com/10_Lib/10_Conv/12_MFCS/11_SIS/FB_SIS_MsgManager_6_1.TcPOU $
 *
 *	Purpose			:	Send GVR
 *
 * ------------------------------------------------------------------------------------
 *	Copyright Swisslog [IP AG], Switzerland. All rights reserved.
 * 
 * ------------------------------------------------------------------------------------
 *	
 * 	Revision History: 
 *
 * 	VERSION			DATE			INITIALS			DESCRIPTION
 *	0.1				01.01.2001		swl					Example
 *
 **************************************************************************************)
VAR_INPUT
 	meChannelSrc		: E_MFCS_Channel; // Source communicaton channel
	mpGVR				: POINTER TO ST_ITC_GVR; // Pointer to GVR
END_VAR
(**************************************************************************************************************
 	Check if a telegram needs to be send
***************************************************************************************************************)
// If settings allow sending a GVR 	
IF  Settings.Telegrams.SendGVR THEN
	// If the source of the request is this channel or is undefined
	IF meChannelSrc = Settings.MFCS_Channel OR
		meChannelSrc = E_MFCS_Channel.BEGIN_CHANNEL THEN
		;//Proceed
	ELSE // Source is a different MFCS Connection
		// Dont send a telegram		
		RETURN;
	END_IF	
ELSE
	// Dont send a telegram		
	RETURN;
END_IF

(**************************************************************************************************************
 	ITC - Map generic data to type
***************************************************************************************************************)
MEMCPY(destAddr := ADR(GVR_ITC), srcAddr := mpGVR, n := SIZEOF(GVR_ITC));

(**************************************************************************************************************
 	Formatting data
***************************************************************************************************************)

// Get Number 
GVR.Number := 	F_StuffString(
					InputString 	:= INT_TO_STRING(GVR_ITC.Number), 
					StringLength	:= SIS_6_1.GVR_NUMBER_STRINGLENGTH, 
					StuffCharacter 	:= '0',
					LeftAligned		:= FALSE);

// Get Quantity 
GVR.Quantity := F_StuffString(
					InputString 	:= INT_TO_STRING(GVR_ITC.Quantity), 
					StringLength	:= SIS_6_1.GVR_QUANTITY_STRINGLENGTH, 
					StuffCharacter 	:= '0',
					LeftAligned		:= FALSE);

// Initialize values
FOR Idx := 0 TO 9 DO
	GVR.Variable[Idx] := '0';
END_FOR

// Fill values
FOR Idx := 0 TO 9 DO
	GVR.Variable[Idx] := F_StuffString(
							InputString 	:= DINT_TO_STRING(GVR_ITC.Variable[Idx]), 
							StringLength	:= SIS_6_1.GVR_VARIABLE_STRINGLENGTH, 
							StuffCharacter 	:= '0',
							LeftAligned		:= FALSE);
	
END_FOR

// Get ReturnCode 
GVR.ReturnCode := F_StuffString(
					InputString 	:= INT_TO_STRING(GVR_ITC.ReturnCode), 
					StringLength	:= SIS_6_1.ERRORCODE_STRINGLENGTH, 
					StuffCharacter 	:= '0',
					LeftAligned		:= FALSE);


(**************************************************************************************************************
 	Build string and add to Base Driver
***************************************************************************************************************)
MEMSET(destAddr := ADR(SendTelegram), 0, SIZEOF(SendTelegram));
WritePointer := 0;

F_AssembleByteStream(
	pSrc:= ADR('GVR'), 
	SrcLen:= 3, 
	pDest:= ADR(SendTelegram), 
	DestLen:= SIZEOF(SendTelegram), 
	WritePointer:= WritePointer);
	
F_AssembleByteStream(
	pSrc:= ADR(GVR.Number), 
	SrcLen:= INT_TO_UDINT(LEN(GVR.Number)), 
	pDest:= ADR(SendTelegram), 
	DestLen:= SIZEOF(SendTelegram), 
	WritePointer:= WritePointer);	

F_AssembleByteStream(
	pSrc:= ADR(GVR.Quantity), 
	SrcLen:= INT_TO_UDINT(LEN(GVR.Quantity)), 
	pDest:= ADR(SendTelegram), 
	DestLen:= SIZEOF(SendTelegram), 
	WritePointer:= WritePointer);	

// Add Variables 
FOR Idx := 0 TO 9 DO
	F_AssembleByteStream(
		pSrc:= ADR(GVR.Variable[Idx]), 
		SrcLen:= INT_TO_UDINT(LEN(GVR.Variable[Idx])), 
		pDest:= ADR(SendTelegram), 
		DestLen:= SIZEOF(SendTelegram), 
		WritePointer:= WritePointer);	
END_FOR

F_AssembleByteStream(
	pSrc:= ADR(GVR.ReturnCode), 
	SrcLen:= INT_TO_UDINT(LEN(GVR.ReturnCode)), 
	pDest:= ADR(SendTelegram), 
	DestLen:= SIZEOF(SendTelegram), 
	WritePointer:= WritePointer);

// Add to buffer of Base Driver
M_ProcessGVR := fbBaseDriver.M_SendAppData(
					mpSendData := ADR(SendTelegram),
					mSendDataLen := WritePointer);

// Forward to mirror channel
M_MirrorData(Data := ADR(SendTelegram), DataLen := WritePointer);
END_METHOD

METHOD PROTECTED M_ProcessIPR : BOOL
(**************************************************************************************
 * 	Application		:	BoxControl Framework
 *	Revision		:	$Revision: 404529 $
 *	Revision date	:	$Date: 2018-04-23 08:21:38 +0200 (Mo., 23 Apr 2018) $
 *	Last changed by	:	$Author: b7bolm $
 *	URL				:	$URL: http://almscdc.swisslog.com/repo/SWPD/Development/BoxControlFramework/20_Release/trunk/01_Software/BCF/BCF/JumpStart/20_Product/10_App/11_Com/10_Lib/10_Conv/12_MFCS/11_SIS/FB_SIS_MsgManager_6_1.TcPOU $
 *
 *	Purpose			:	Send IPR
 *
 * ------------------------------------------------------------------------------------
 *	Copyright Swisslog [IP AG], Switzerland. All rights reserved.
 * 
 * ------------------------------------------------------------------------------------
 *	
 * 	Revision History: 
 *
 * 	VERSION			DATE			INITIALS			DESCRIPTION
 *	0.1				01.01.2001		swl					Example
 *
 **************************************************************************************)
VAR_INPUT
 	meChannelSrc		: E_MFCS_Channel; // Source communicaton channel
	mpIPR				: POINTER TO ST_ITC_IPR; // Pointer to IPR
END_VAR
(**************************************************************************************************************
 	Check if a telegram needs to be send
***************************************************************************************************************)
// If settings allow sending a IPR 	
IF  Settings.Telegrams.SendIPR THEN
	// If the source of the request is this channel or is undefined
	IF meChannelSrc = Settings.MFCS_Channel OR
		meChannelSrc = E_MFCS_Channel.BEGIN_CHANNEL THEN
		;//Proceed
	ELSE // Source is a different MFCS Connection
		// Dont send a telegram		
		RETURN;
	END_IF	
ELSE
	// Dont send a telegram		
	RETURN;
END_IF

(**************************************************************************************************************
 	ITC - Map generic data to type
***************************************************************************************************************)
MEMCPY(destAddr := ADR(IPR_ITC), srcAddr := mpIPR, n := SIZEOF(IPR_ITC));


(**************************************************************************************************************
 	Formatting data
***************************************************************************************************************)

// Get SIS-Number 
IPR.Position := F_StuffString(
					InputString 	:= IPR_ITC.Position, 
					StringLength	:= SIS_6_1.POSITION_STRINGLENGTH, 
					StuffCharacter 	:= '0',
					LeftAligned		:= FALSE);

// Get TU-DataIndex 
IPR.TU_DataIndex := F_StuffString(
						InputString 	:= DINT_TO_STRING(IPR_ITC.TU_DataIndex), 
						StringLength	:= SIS_6_1.TU_DATAINDEX_STRINGLENGTH, 
						StuffCharacter 	:= '0',
						LeftAligned		:= FALSE);

// Get MSG Sequence 
IPR.MSG_Sequence := F_StuffString(
						InputString 	:= INT_TO_STRING(IPR_ITC.MSG_Sequence), 
						StringLength	:= SIS_6_1.MSG_SEQUENCE_STRINGLENGTH, 
						StuffCharacter 	:= '0',
						LeftAligned		:= FALSE);

// Get TU-ID 
IPR.TU_ID := F_StuffString(
				InputString 	:= IPR_ITC.TU_ID, 
				StringLength	:= SIS_6_1.TU_ID_STRINGLENGTH, 
				StuffCharacter 	:= ' ',
				LeftAligned		:= FALSE);

// Get TU-Type 
IPR.TU_Type := F_StuffString(
				InputString 	:= INT_TO_STRING(IPR_ITC.TU_Type), 
				StringLength	:= SIS_6_1.TU_TYPE_STRINGLENGTH, 
				StuffCharacter 	:= '0',
				LeftAligned		:= FALSE);			

// Get Assignment id 
IPR.AssignmentID := F_StuffString(
						InputString 	:= UDINT_TO_STRING(IPR_ITC.AssignmentID), 
						StringLength	:= SIS_6_1.ASSIGNMENT_ID_STRINGLENGTH, 
						StuffCharacter 	:= '0',
						LeftAligned		:= FALSE);
				
// Get Height
IPR.Height := F_StuffString(
						InputString 	:= INT_TO_STRING(IPR_ITC.Height), 
						StringLength	:= SIS_6_1.IPR_HEIGHT_STRINGLENGTH, 
						StuffCharacter 	:= '0',
						LeftAligned		:= FALSE);;
				
// Get Width Right 
IPR.WidthRight := F_StuffString(
						InputString 	:= INT_TO_STRING(IPR_ITC.WidthRight), 
						StringLength	:= SIS_6_1.IPR_WIDTHRIGHT_STRINGLENGTH, 
						StuffCharacter 	:= '0',
						LeftAligned		:= FALSE);
				
// Get Width Left 
IPR.WidthLeft := F_StuffString(
						InputString 	:= INT_TO_STRING(IPR_ITC.WidthLeft), 
						StringLength	:= SIS_6_1.IPR_WIDTHLEFT_STRINGLENGTH, 
						StuffCharacter 	:= '0',
						LeftAligned		:= FALSE);	
						
// Get Length Front 
IPR.LengthFront := F_StuffString(
						InputString 	:= INT_TO_STRING(IPR_ITC.LengthFront), 
						StringLength	:= SIS_6_1.IPR_LENGTHFRONT_STRINGLENGTH, 
						StuffCharacter 	:= '0',
						LeftAligned		:= FALSE);
						
// Get Length Rear 
IPR.LengthRear := F_StuffString(
						InputString 	:= INT_TO_STRING(IPR_ITC.LengthRear), 
						StringLength	:= SIS_6_1.IPR_LENGTHREAR_STRINGLENGTH, 
						StuffCharacter 	:= '0',
						LeftAligned		:= FALSE);

// Get Weight 
IPR.Weight := F_StuffString(
				InputString 	:= DINT_TO_STRING(IPR_ITC.Weight), 
				StringLength	:= SIS_6_1.IPR_WEIGHT_STRINGLENGTH, 
				StuffCharacter 	:= '0',
				LeftAligned		:= FALSE);

// Get Tunnel 
IPR.Tunnel := INT_TO_STRING(IPR_ITC.Tunnel);

// Get Runner 
IPR.Runner := INT_TO_STRING(IPR_ITC.Runner);

// Get Error 
IPR.ErrorCode := F_StuffString(
					InputString 	:= INT_TO_STRING(IPR_ITC.ErrorCode), 
					StringLength	:= SIS_6_1.ERRORCODE_STRINGLENGTH, 
					StuffCharacter 	:= '0',
					LeftAligned		:= FALSE);


// Get Valid Label String 
IPR.ValidLabelString := F_StuffString(
							InputString 	:= INT_TO_STRING(IPR_ITC.ValidLabelString), 
							StringLength	:= SIS_6_1.IPR_VALIDLABELSTRING_STRINGLENGTH, 
							StuffCharacter 	:= '0',
							LeftAligned		:= FALSE);

// Get Label 
IPR.Label:= F_StuffString(
				InputString 	:= IPR_ITC.Label, 
				StringLength	:= Conveyor.LABEL_LENGTH, 
				StuffCharacter 	:= '-',
				LeftAligned		:= FALSE);


(**************************************************************************************************************
 	Build string and add to Base Driver
***************************************************************************************************************)
MEMSET(destAddr := ADR(SendTelegram), 0, SIZEOF(SendTelegram));
WritePointer := 0;

F_AssembleByteStream(
	pSrc:= ADR('IPR'), 
	SrcLen:= 3, 
	pDest:= ADR(SendTelegram), 
	DestLen:= SIZEOF(SendTelegram), 
	WritePointer:= WritePointer);
	
F_AssembleByteStream(
	pSrc:= ADR(IPR.Position), 
	SrcLen:= INT_TO_UDINT(LEN(IPR.Position)), 
	pDest:= ADR(SendTelegram), 
	DestLen:= SIZEOF(SendTelegram), 
	WritePointer:= WritePointer);
	
F_AssembleByteStream(
	pSrc:= ADR(IPR.TU_DataIndex), 
	SrcLen:= INT_TO_UDINT(LEN(IPR.TU_DataIndex)), 
	pDest:= ADR(SendTelegram), 
	DestLen:= SIZEOF(SendTelegram), 
	WritePointer:= WritePointer);
	
F_AssembleByteStream(
	pSrc:= ADR(IPR.MSG_Sequence), 
	SrcLen:= INT_TO_UDINT(LEN(IPR.MSG_Sequence)), 
	pDest:= ADR(SendTelegram), 
	DestLen:= SIZEOF(SendTelegram), 
	WritePointer:= WritePointer);

F_AssembleByteStream(
	pSrc:= ADR(IPR.TU_ID), 
	SrcLen:= INT_TO_UDINT(LEN(IPR.TU_ID)), 
	pDest:= ADR(SendTelegram), 
	DestLen:= SIZEOF(SendTelegram), 
	WritePointer:= WritePointer);

F_AssembleByteStream(
	pSrc:= ADR(IPR.TU_Type), 
	SrcLen:= INT_TO_UDINT(LEN(IPR.TU_Type)), 
	pDest:= ADR(SendTelegram), 
	DestLen:= SIZEOF(SendTelegram), 
	WritePointer:= WritePointer);

F_AssembleByteStream(
	pSrc:= ADR(IPR.AssignmentID), 
	SrcLen:= INT_TO_UDINT(LEN(IPR.AssignmentID)), 
	pDest:= ADR(SendTelegram), 
	DestLen:= SIZEOF(SendTelegram), 
	WritePointer:= WritePointer);

F_AssembleByteStream(
	pSrc:= ADR(IPR.Height), 
	SrcLen:= INT_TO_UDINT(LEN(IPR.Height)), 
	pDest:= ADR(SendTelegram), 
	DestLen:= SIZEOF(SendTelegram), 
	WritePointer:= WritePointer);

F_AssembleByteStream(
	pSrc:= ADR(IPR.WidthRight), 
	SrcLen:= INT_TO_UDINT(LEN(IPR.WidthRight)), 
	pDest:= ADR(SendTelegram), 
	DestLen:= SIZEOF(SendTelegram), 
	WritePointer:= WritePointer);

F_AssembleByteStream(
	pSrc:= ADR(IPR.WidthLeft), 
	SrcLen:= INT_TO_UDINT(LEN(IPR.WidthLeft)), 
	pDest:= ADR(SendTelegram), 
	DestLen:= SIZEOF(SendTelegram), 
	WritePointer:= WritePointer);

F_AssembleByteStream(
	pSrc:= ADR(IPR.LengthFront), 
	SrcLen:= INT_TO_UDINT(LEN(IPR.LengthFront)), 
	pDest:= ADR(SendTelegram), 
	DestLen:= SIZEOF(SendTelegram), 
	WritePointer:= WritePointer);

F_AssembleByteStream(
	pSrc:= ADR(IPR.LengthRear), 
	SrcLen:= INT_TO_UDINT(LEN(IPR.LengthRear)), 
	pDest:= ADR(SendTelegram), 
	DestLen:= SIZEOF(SendTelegram), 
	WritePointer:= WritePointer);

F_AssembleByteStream(
	pSrc:= ADR(IPR.Weight), 
	SrcLen:= INT_TO_UDINT(LEN(IPR.Weight)), 
	pDest:= ADR(SendTelegram), 
	DestLen:= SIZEOF(SendTelegram), 
	WritePointer:= WritePointer);

F_AssembleByteStream(
	pSrc:= ADR(IPR.Tunnel), 
	SrcLen:= INT_TO_UDINT(LEN(IPR.Tunnel)), 
	pDest:= ADR(SendTelegram), 
	DestLen:= SIZEOF(SendTelegram), 
	WritePointer:= WritePointer);

F_AssembleByteStream(
	pSrc:= ADR(IPR.Runner), 
	SrcLen:= INT_TO_UDINT(LEN(IPR.Runner)), 
	pDest:= ADR(SendTelegram), 
	DestLen:= SIZEOF(SendTelegram), 
	WritePointer:= WritePointer);

F_AssembleByteStream(
	pSrc:= ADR(IPR.ErrorCode), 
	SrcLen:= INT_TO_UDINT(LEN(IPR.ErrorCode)), 
	pDest:= ADR(SendTelegram), 
	DestLen:= SIZEOF(SendTelegram), 
	WritePointer:= WritePointer);

F_AssembleByteStream(
	pSrc:= ADR(IPR.ValidLabelString), 
	SrcLen:= INT_TO_UDINT(LEN(IPR.ValidLabelString)), 
	pDest:= ADR(SendTelegram), 
	DestLen:= SIZEOF(SendTelegram), 
	WritePointer:= WritePointer);

F_AssembleByteStream(
	pSrc:= ADR(IPR.Label), 
	SrcLen:= INT_TO_UDINT(LEN(IPR.Label)), 
	pDest:= ADR(SendTelegram), 
	DestLen:= SIZEOF(SendTelegram), 
	WritePointer:= WritePointer);

// Add to buffer of Base Driver
M_ProcessIPR := fbBaseDriver.M_SendAppData(
					mpSendData := ADR(SendTelegram),
					mSendDataLen := WritePointer);

// Forward to mirror channel
M_MirrorData(Data := ADR(SendTelegram), DataLen := WritePointer);
END_METHOD

METHOD PROTECTED M_ProcessISR : BOOL
(**************************************************************************************
 * 	Application		:	BoxControl Framework
 *	Revision		:	$Revision: 404529 $
 *	Revision date	:	$Date: 2018-04-23 08:21:38 +0200 (Mo., 23 Apr 2018) $
 *	Last changed by	:	$Author: b7bolm $
 *	URL				:	$URL: http://almscdc.swisslog.com/repo/SWPD/Development/BoxControlFramework/20_Release/trunk/01_Software/BCF/BCF/JumpStart/20_Product/10_App/11_Com/10_Lib/10_Conv/12_MFCS/11_SIS/FB_SIS_MsgManager_6_1.TcPOU $
 *
 *	Purpose			:	Send ISR
 *
 * ------------------------------------------------------------------------------------
 *	Copyright Swisslog [IP AG], Switzerland. All rights reserved.
 * 
 * ------------------------------------------------------------------------------------
 *	
 * 	Revision History: 
 *
 * 	VERSION			DATE			INITIALS			DESCRIPTION
 *	0.1				01.01.2001		swl					Example
 *
 **************************************************************************************)
VAR_INPUT
 	meChannelSrc		: E_MFCS_Channel; // Source communicaton channel
	mpISR				: POINTER TO ST_ITC_ISR; // Pointer to ISR
END_VAR

VAR
	Idx					: INT; // Iterator
	TempByte			: BYTE; // Temporary byte
	TempInt				: INT; // Temporary int
END_VAR
(**************************************************************************************************************
 	Check if a telegram needs to be send
***************************************************************************************************************)
// If settings allow sending a ISR 	
IF  Settings.Telegrams.SendISR THEN
	// If the source of the request is this channel or is undefined
	IF meChannelSrc = Settings.MFCS_Channel OR
		meChannelSrc = E_MFCS_Channel.BEGIN_CHANNEL THEN
		;//Proceed
	ELSE // Source is a different MFCS Connection
		// Dont send a telegram		
		RETURN;
	END_IF	
ELSE
	// Dont send a telegram		
	RETURN;
END_IF

(**************************************************************************************************************
 	ITC - Map generic data to type
***************************************************************************************************************)
MEMCPY(destAddr := ADR(ISR_ITC), srcAddr := mpISR, n := SIZEOF(ISR_ITC));

(**************************************************************************************************************
 	Formatting data
***************************************************************************************************************)

// Set the ISR.SignalType 
ISR.SignalType := INT_TO_STRING(ISR_ITC.SignalType);

// Set the ISR.StartingSignalNumber 
ISR.StartSignalNumber := F_StuffString(
							InputString 	:= INT_TO_STRING(ISR_ITC.StartSignalNumber), 
							StringLength	:= SIS_6_1.ISR_SIGNALNUMBER_STRINGLENGTH, 
							StuffCharacter 	:= '0',
						LeftAligned		:= FALSE);

// Set the ISR.DataLength 
ISR.DataLength := F_StuffString(
							InputString 	:= INT_TO_STRING(ISR_ITC.DataLength), 
							StringLength	:= SIS_6_1.ISR_DATALENGTH_STRINGLENGTH, 
							StuffCharacter 	:= '0',
						LeftAligned		:= FALSE);

// Store information
ISR.Information	:= ISR_ITC.Information;

ISR.ReturnCode := F_StuffString(
					InputString 	:= INT_TO_STRING(ISR_ITC.ReturnCode), 
					StringLength	:= SIS_6_1.ERRORCODE_STRINGLENGTH, 
					StuffCharacter 	:= '0',
					LeftAligned		:= FALSE);
							
(**************************************************************************************************************
 	Build string and add to Base Driver
***************************************************************************************************************)
MEMSET(destAddr := ADR(SendTelegram), 0, SIZEOF(SendTelegram));
WritePointer := 0;

F_AssembleByteStream(
	pSrc:= ADR('ISR'), 
	SrcLen:= 3, 
	pDest:= ADR(SendTelegram), 
	DestLen:= SIZEOF(SendTelegram), 
	WritePointer:= WritePointer);
	
F_AssembleByteStream(
	pSrc:= ADR(ISR.SignalType), 
	SrcLen:= INT_TO_UDINT(LEN(ISR.SignalType)), 
	pDest:= ADR(SendTelegram), 
	DestLen:= SIZEOF(SendTelegram), 
	WritePointer:= WritePointer);

F_AssembleByteStream(
	pSrc:= ADR(ISR.StartSignalNumber), 
	SrcLen:= INT_TO_UDINT(LEN(ISR.StartSignalNumber)), 
	pDest:= ADR(SendTelegram), 
	DestLen:= SIZEOF(SendTelegram), 
	WritePointer:= WritePointer);

F_AssembleByteStream(
	pSrc:= ADR(ISR.DataLength), 
	SrcLen:= INT_TO_UDINT(LEN(ISR.DataLength)), 
	pDest:= ADR(SendTelegram), 
	DestLen:= SIZEOF(SendTelegram), 
	WritePointer:= WritePointer);

F_AssembleByteStream(
	pSrc:= ADR(ISR.Information), 
	SrcLen:= INT_TO_UDINT(LEN(ISR.Information)), 
	pDest:= ADR(SendTelegram), 
	DestLen:= SIZEOF(SendTelegram), 
	WritePointer:= WritePointer);

F_AssembleByteStream(
	pSrc:= ADR(ISR.ReturnCode), 
	SrcLen:= INT_TO_UDINT(LEN(ISR.ReturnCode)), 
	pDest:= ADR(SendTelegram), 
	DestLen:= SIZEOF(SendTelegram), 
	WritePointer:= WritePointer);

// Add to buffer of Base Driver
M_ProcessISR := fbBaseDriver.M_SendAppData(
					mpSendData := ADR(SendTelegram),
					mSendDataLen := WritePointer);

// Forward to mirror channel
M_MirrorData(Data := ADR(SendTelegram), DataLen := WritePointer);
END_METHOD

METHOD PROTECTED M_ProcessMCR : BOOL
(**************************************************************************************
 * 	Application		:	BoxControl Framework
 *	Revision		:	$Revision: 404529 $
 *	Revision date	:	$Date: 2018-04-23 08:21:38 +0200 (Mo., 23 Apr 2018) $
 *	Last changed by	:	$Author: b7bolm $
 *	URL				:	$URL: http://almscdc.swisslog.com/repo/SWPD/Development/BoxControlFramework/20_Release/trunk/01_Software/BCF/BCF/JumpStart/20_Product/10_App/11_Com/10_Lib/10_Conv/12_MFCS/11_SIS/FB_SIS_MsgManager_6_1.TcPOU $
 *
 *	Purpose			:	Send MCR
 *
 * ------------------------------------------------------------------------------------
 *	Copyright Swisslog [IP AG], Switzerland. All rights reserved.
 * 
 * ------------------------------------------------------------------------------------
 *	
 * 	Revision History: 
 *
 * 	VERSION			DATE			INITIALS			DESCRIPTION
 *	0.1				01.01.2001		swl					Example
 *
 **************************************************************************************)
VAR_INPUT
 	meChannelSrc		: E_MFCS_Channel; // Source communicaton channel
	mpMCR				: POINTER TO ST_ITC_MCR; // Pointer to MCR
END_VAR
(**************************************************************************************************************
 	Check if a telegram needs to be send
***************************************************************************************************************)
// If settings allow sending a MCR 	
IF  Settings.Telegrams.SendMCR THEN
	// If the source of the request is this channel or is undefined
	IF meChannelSrc = Settings.MFCS_Channel OR
		meChannelSrc = E_MFCS_Channel.BEGIN_CHANNEL THEN
		;//Proceed
	ELSE // Source is a different MFCS Connection
		// Dont send a telegram		
		RETURN;
	END_IF	
ELSE
	// Dont send a telegram		
	RETURN;
END_IF

(**************************************************************************************************************
 	ITC - Map generic data to type
***************************************************************************************************************)
MEMCPY(destAddr := ADR(MCR_ITC), srcAddr := mpMCR, n := SIZEOF(MCR_ITC));

(**************************************************************************************************************
 	Formatting data
***************************************************************************************************************)

// Get position
MCR.Position := F_StuffString(
					InputString 	:= MCR_ITC.Position, 
					StringLength	:= SIS_6_1.POSITION_STRINGLENGTH, 
					StuffCharacter 	:= '0',
					LeftAligned		:= FALSE);;
					
// Get Code 
MCR.Code := F_StuffString(
				InputString 	:= INT_TO_STRING(MCR_ITC.Code), 
				StringLength	:= SIS_6_1.MCR_CODE_STRINGLENGTH, 
				StuffCharacter 	:= '0',
				LeftAligned		:= FALSE);

// Get mode
MCR.Mode := INT_TO_STRING(MCR_ITC.Mode);

// Get speed
IF MCR_ITC.Speed.Enable THEN
	IF MCR_ITC.Speed.Fast THEN
		MCR.Speed := '2';
	ELSE
		MCR.Speed := '1';
	END_IF
ELSE
	MCR.Speed := '0';
END_IF


// Get Axis fwd
IF MCR_ITC.Axis[1].Forward.Enable THEN
	IF MCR_ITC.Axis[1].Forward.Selected THEN
		MCR.Axis1Fwd := '2';
	ELSE
		MCR.Axis1Fwd := '1';
	END_IF
ELSE
	MCR.Axis1Fwd := '0';
END_IF

// Get Axis rev
IF MCR_ITC.Axis[1].Reverse.Enable THEN
	IF MCR_ITC.Axis[1].Reverse.Selected THEN
		MCR.Axis1Rev := '2';
	ELSE
		MCR.Axis1Rev := '1';
	END_IF
ELSE
	MCR.Axis1Rev := '0';
END_IF

// Get Axis fwd
IF MCR_ITC.Axis[2].Forward.Enable THEN
	IF MCR_ITC.Axis[2].Forward.Selected THEN
		MCR.Axis2Fwd := '2';
	ELSE
		MCR.Axis2Fwd := '1';
	END_IF
ELSE
	MCR.Axis2Fwd := '0';
END_IF

// Get Axis rev
IF MCR_ITC.Axis[2].Reverse.Enable THEN
	IF MCR_ITC.Axis[2].Reverse.Selected THEN
		MCR.Axis2Rev := '2';
	ELSE
		MCR.Axis2Rev := '1';
	END_IF
ELSE
	MCR.Axis2Rev := '0';
END_IF

// Get Axis fwd
IF MCR_ITC.Axis[3].Forward.Enable THEN
	IF MCR_ITC.Axis[3].Forward.Selected THEN
		MCR.Axis3Fwd := '2';
	ELSE
		MCR.Axis3Fwd := '1';
	END_IF
ELSE
	MCR.Axis3Fwd := '0';
END_IF

// Get Axis rev
IF MCR_ITC.Axis[3].Reverse.Enable THEN
	IF MCR_ITC.Axis[3].Reverse.Selected THEN
		MCR.Axis3Rev := '2';
	ELSE
		MCR.Axis3Rev := '1';
	END_IF
ELSE
	MCR.Axis3Rev := '0';
END_IF

// Get Axis fwd
IF MCR_ITC.Axis[4].Forward.Enable THEN
	IF MCR_ITC.Axis[4].Forward.Selected THEN
		MCR.Axis4Fwd := '2';
	ELSE
		MCR.Axis4Fwd := '1';
	END_IF
ELSE
	MCR.Axis4Fwd := '0';
END_IF

// Get Axis rev
IF MCR_ITC.Axis[4].Reverse.Enable THEN
	IF MCR_ITC.Axis[4].Reverse.Selected THEN
		MCR.Axis4Rev := '2';
	ELSE
		MCR.Axis4Rev := '1';
	END_IF
ELSE
	MCR.Axis4Rev := '0';
END_IF

// Get Axis fwd
IF MCR_ITC.Axis[5].Forward.Enable THEN
	IF MCR_ITC.Axis[5].Forward.Selected THEN
		MCR.Axis5Fwd := '2';
	ELSE
		MCR.Axis5Fwd := '1';
	END_IF
ELSE
	MCR.Axis5Fwd := '0';
END_IF

// Get Axis rev
IF MCR_ITC.Axis[5].Reverse.Enable THEN
	IF MCR_ITC.Axis[5].Reverse.Selected THEN
		MCR.Axis5Rev := '2';
	ELSE
		MCR.Axis5Rev := '1';
	END_IF
ELSE
	MCR.Axis5Rev := '0';
END_IF

// Get Axis fwd
IF MCR_ITC.Axis[6].Forward.Enable THEN
	IF MCR_ITC.Axis[6].Forward.Selected THEN
		MCR.Axis6Fwd := '2';
	ELSE
		MCR.Axis6Fwd := '1';
	END_IF
ELSE
	MCR.Axis6Fwd := '0';
END_IF

// Get Axis rev
IF MCR_ITC.Axis[6].Reverse.Enable THEN
	IF MCR_ITC.Axis[6].Reverse.Selected THEN
		MCR.Axis6Rev := '2';
	ELSE
		MCR.Axis6Rev := '1';
	END_IF
ELSE
	MCR.Axis6Rev := '0';
END_IF

// Get Button 1
IF MCR_ITC.Button[1].Enable THEN
	IF MCR_ITC.Button[1].Selected THEN
		MCR.Button1 := '2';
	ELSE
		MCR.Button1 := '1';
	END_IF
ELSE
	MCR.Button1 := '0';
END_IF

// Get Button 2
IF MCR_ITC.Button[2].Enable THEN
	IF MCR_ITC.Button[2].Selected THEN
		MCR.Button2 := '2';
	ELSE
		MCR.Button2 := '1';
	END_IF
ELSE
	MCR.Button2 := '0';
END_IF

// Get return code
MCR.ReturnCode := F_StuffString(
					InputString 	:= INT_TO_STRING(MCR_ITC.eReturnCode), 
					StringLength	:= SIS_6_1.ERRORCODE_STRINGLENGTH, 
					StuffCharacter 	:= '0',
					LeftAligned		:= FALSE);

(**************************************************************************************************************
 	Build string and add to Base Driver
***************************************************************************************************************)
MEMSET(destAddr := ADR(SendTelegram), 0, SIZEOF(SendTelegram));
WritePointer := 0;

F_AssembleByteStream(
	pSrc:= ADR('MCR'), 
	SrcLen:= 3, 
	pDest:= ADR(SendTelegram), 
	DestLen:= SIZEOF(SendTelegram), 
	WritePointer:= WritePointer);
	
F_AssembleByteStream(
	pSrc:= ADR(MCR.Position), 
	SrcLen:= INT_TO_UDINT(LEN(MCR.Position)), 
	pDest:= ADR(SendTelegram), 
	DestLen:= SIZEOF(SendTelegram), 
	WritePointer:= WritePointer);

F_AssembleByteStream(
	pSrc:= ADR(MCR.Code), 
	SrcLen:= INT_TO_UDINT(LEN(MCR.Code)), 
	pDest:= ADR(SendTelegram), 
	DestLen:= SIZEOF(SendTelegram), 
	WritePointer:= WritePointer);

F_AssembleByteStream(
	pSrc:= ADR(MCR.Mode), 
	SrcLen:= INT_TO_UDINT(LEN(MCR.Mode)), 
	pDest:= ADR(SendTelegram), 
	DestLen:= SIZEOF(SendTelegram), 
	WritePointer:= WritePointer);

F_AssembleByteStream(
	pSrc:= ADR(MCR.Speed), 
	SrcLen:= INT_TO_UDINT(LEN(MCR.Speed)), 
	pDest:= ADR(SendTelegram), 
	DestLen:= SIZEOF(SendTelegram), 
	WritePointer:= WritePointer);

F_AssembleByteStream(
	pSrc:= ADR(MCR.Axis1Fwd), 
	SrcLen:= INT_TO_UDINT(LEN(MCR.Axis1Fwd)), 
	pDest:= ADR(SendTelegram), 
	DestLen:= SIZEOF(SendTelegram), 
	WritePointer:= WritePointer);

F_AssembleByteStream(
	pSrc:= ADR(MCR.Axis1Rev), 
	SrcLen:= INT_TO_UDINT(LEN(MCR.Axis1Rev)), 
	pDest:= ADR(SendTelegram), 
	DestLen:= SIZEOF(SendTelegram), 
	WritePointer:= WritePointer);

F_AssembleByteStream(
	pSrc:= ADR(MCR.Axis2Fwd), 
	SrcLen:= INT_TO_UDINT(LEN(MCR.Axis2Fwd)), 
	pDest:= ADR(SendTelegram), 
	DestLen:= SIZEOF(SendTelegram), 
	WritePointer:= WritePointer);

F_AssembleByteStream(
	pSrc:= ADR(MCR.Axis2Rev), 
	SrcLen:= INT_TO_UDINT(LEN(MCR.Axis2Rev)), 
	pDest:= ADR(SendTelegram), 
	DestLen:= SIZEOF(SendTelegram), 
	WritePointer:= WritePointer);

F_AssembleByteStream(
	pSrc:= ADR(MCR.Axis3Fwd), 
	SrcLen:= INT_TO_UDINT(LEN(MCR.Axis3Fwd)), 
	pDest:= ADR(SendTelegram), 
	DestLen:= SIZEOF(SendTelegram), 
	WritePointer:= WritePointer);

F_AssembleByteStream(
	pSrc:= ADR(MCR.Axis3Rev), 
	SrcLen:= INT_TO_UDINT(LEN(MCR.Axis3Rev)), 
	pDest:= ADR(SendTelegram), 
	DestLen:= SIZEOF(SendTelegram), 
	WritePointer:= WritePointer);

F_AssembleByteStream(
	pSrc:= ADR(MCR.Axis4Fwd), 
	SrcLen:= INT_TO_UDINT(LEN(MCR.Axis4Fwd)), 
	pDest:= ADR(SendTelegram), 
	DestLen:= SIZEOF(SendTelegram), 
	WritePointer:= WritePointer);

F_AssembleByteStream(
	pSrc:= ADR(MCR.Axis4Rev), 
	SrcLen:= INT_TO_UDINT(LEN(MCR.Axis4Rev)), 
	pDest:= ADR(SendTelegram), 
	DestLen:= SIZEOF(SendTelegram), 
	WritePointer:= WritePointer);
	
F_AssembleByteStream(
	pSrc:= ADR(MCR.Axis5Fwd), 
	SrcLen:= INT_TO_UDINT(LEN(MCR.Axis5Fwd)), 
	pDest:= ADR(SendTelegram), 
	DestLen:= SIZEOF(SendTelegram), 
	WritePointer:= WritePointer);

F_AssembleByteStream(
	pSrc:= ADR(MCR.Axis5Rev), 
	SrcLen:= INT_TO_UDINT(LEN(MCR.Axis5Rev)), 
	pDest:= ADR(SendTelegram), 
	DestLen:= SIZEOF(SendTelegram), 
	WritePointer:= WritePointer);

F_AssembleByteStream(
	pSrc:= ADR(MCR.Axis6Fwd), 
	SrcLen:= INT_TO_UDINT(LEN(MCR.Axis6Fwd)), 
	pDest:= ADR(SendTelegram), 
	DestLen:= SIZEOF(SendTelegram), 
	WritePointer:= WritePointer);

F_AssembleByteStream(
	pSrc:= ADR(MCR.Axis6Rev), 
	SrcLen:= INT_TO_UDINT(LEN(MCR.Axis6Rev)), 
	pDest:= ADR(SendTelegram), 
	DestLen:= SIZEOF(SendTelegram), 
	WritePointer:= WritePointer);

F_AssembleByteStream(
	pSrc:= ADR(MCR.Button1), 
	SrcLen:= INT_TO_UDINT(LEN(MCR.Button1)), 
	pDest:= ADR(SendTelegram), 
	DestLen:= SIZEOF(SendTelegram), 
	WritePointer:= WritePointer);	
	
F_AssembleByteStream(
	pSrc:= ADR(MCR.Button2), 
	SrcLen:= INT_TO_UDINT(LEN(MCR.Button2)), 
	pDest:= ADR(SendTelegram), 
	DestLen:= SIZEOF(SendTelegram), 
	WritePointer:= WritePointer);	
	
F_AssembleByteStream(
	pSrc:= ADR(MCR.ReturnCode), 
	SrcLen:= INT_TO_UDINT(LEN(MCR.ReturnCode)), 
	pDest:= ADR(SendTelegram), 
	DestLen:= SIZEOF(SendTelegram), 
	WritePointer:= WritePointer);	


// Add to buffer of Base Driver
M_ProcessMCR := fbBaseDriver.M_SendAppData(
					mpSendData := ADR(SendTelegram),
					mSendDataLen := WritePointer);

// Forward to mirror channel
M_MirrorData(Data := ADR(SendTelegram), DataLen := WritePointer);
END_METHOD

METHOD PROTECTED M_ProcessPOR : BOOL
(**************************************************************************************
 * 	Application		:	BoxControl Framework
 *	Revision		:	$Revision: 404529 $
 *	Revision date	:	$Date: 2018-04-23 08:21:38 +0200 (Mo., 23 Apr 2018) $
 *	Last changed by	:	$Author: b7bolm $
 *	URL				:	$URL: http://almscdc.swisslog.com/repo/SWPD/Development/BoxControlFramework/20_Release/trunk/01_Software/BCF/BCF/JumpStart/20_Product/10_App/11_Com/10_Lib/10_Conv/12_MFCS/11_SIS/FB_SIS_MsgManager_6_1.TcPOU $
 *
 *	Purpose			:	Send POR
 *
 * ------------------------------------------------------------------------------------
 *	Copyright Swisslog [IP AG], Switzerland. All rights reserved.
 * 
 * ------------------------------------------------------------------------------------
 *	
 * 	Revision History: 
 *
 * 	VERSION			DATE			INITIALS			DESCRIPTION
 *	0.1				01.01.2001		swl					Example
 *
 **************************************************************************************)
VAR_INPUT
 	meChannelSrc		: E_MFCS_Channel; // Source communicaton channel
	mpPOR				: POINTER TO ST_ITC_POR; // Pointer to POR
END_VAR
(**************************************************************************************************************
 	Check if a telegram needs to be send
***************************************************************************************************************)
// If settings allow sending a POR 	
IF  Settings.Telegrams.SendPOR THEN
	// If the source of the request is this channel or is undefined
	IF meChannelSrc = Settings.MFCS_Channel OR
		meChannelSrc = E_MFCS_Channel.BEGIN_CHANNEL THEN
		;//Proceed
	ELSE // Source is a different MFCS Connection
		// Dont send a telegram		
		RETURN;
	END_IF	
ELSE
	// Dont send a telegram		
	RETURN;
END_IF

(**************************************************************************************************************
 	ITC - Map generic data to type
***************************************************************************************************************)
MEMCPY(destAddr := ADR(POR_ITC), srcAddr := mpPOR, n := SIZEOF(POR_ITC));

(**************************************************************************************************************
 	Formatting data
***************************************************************************************************************)

// Get SIS-Number 
POR.Position := F_StuffString(
					InputString 	:= POR_ITC.Position, 
					StringLength	:= SIS_6_1.POSITION_STRINGLENGTH, 
					StuffCharacter 	:= '0',
					LeftAligned		:= FALSE);

// Get TU-ID 
POR.TU_ID := F_StuffString(
					InputString 	:= POR_ITC.TU_ID, 
					StringLength	:= SIS_6_1.TU_ID_STRINGLENGTH, 
					StuffCharacter 	:= ' ',
					LeftAligned		:= FALSE);

// Get TU-Type 
POR.TU_Type := F_StuffString(
					InputString 	:= INT_TO_STRING(POR_ITC.TU_Type), 
					StringLength	:= SIS_6_1.TU_TYPE_STRINGLENGTH, 
					StuffCharacter 	:= '0',
					LeftAligned		:= FALSE);
					
// Get Assignment 
POR.AssignmentID := F_StuffString(
						InputString 	:= UDINT_TO_STRING(POR_ITC.AssignmentID), 
						StringLength	:= SIS_6_1.ASSIGNMENT_ID_STRINGLENGTH, 
						StuffCharacter 	:= '0',
						LeftAligned		:= FALSE);

// Get Load Information 
POR.LoadInformation := INT_TO_STRING(BOOL_TO_INT(POR_ITC.LoadInformation));


(**************************************************************************************************************
 	Build string and add to Base Driver
***************************************************************************************************************)
MEMSET(destAddr := ADR(SendTelegram), 0, SIZEOF(SendTelegram));
WritePointer := 0;

F_AssembleByteStream(
	pSrc:= ADR('POR'), 
	SrcLen:= 3, 
	pDest:= ADR(SendTelegram), 
	DestLen:= SIZEOF(SendTelegram), 
	WritePointer:= WritePointer);
	
F_AssembleByteStream(
	pSrc:= ADR(POR.Position), 
	SrcLen:= INT_TO_UDINT(LEN(POR.Position)), 
	pDest:= ADR(SendTelegram), 
	DestLen:= SIZEOF(SendTelegram), 
	WritePointer:= WritePointer);
	
F_AssembleByteStream(
	pSrc:= ADR(POR.TU_ID), 
	SrcLen:= INT_TO_UDINT(LEN(POR.TU_ID)), 
	pDest:= ADR(SendTelegram), 
	DestLen:= SIZEOF(SendTelegram), 
	WritePointer:= WritePointer);	
	
F_AssembleByteStream(
	pSrc:= ADR(POR.TU_Type), 
	SrcLen:= INT_TO_UDINT(LEN(POR.TU_Type)), 
	pDest:= ADR(SendTelegram), 
	DestLen:= SIZEOF(SendTelegram), 
	WritePointer:= WritePointer);	
	
F_AssembleByteStream(
	pSrc:= ADR(POR.AssignmentID), 
	SrcLen:= INT_TO_UDINT(LEN(POR.AssignmentID)), 
	pDest:= ADR(SendTelegram), 
	DestLen:= SIZEOF(SendTelegram), 
	WritePointer:= WritePointer);	
	
F_AssembleByteStream(
	pSrc:= ADR(POR.LoadInformation), 
	SrcLen:= INT_TO_UDINT(LEN(POR.LoadInformation)), 
	pDest:= ADR(SendTelegram), 
	DestLen:= SIZEOF(SendTelegram), 
	WritePointer:= WritePointer);	

// Add to buffer of Base Driver
M_ProcessPOR := fbBaseDriver.M_SendAppData(
					mpSendData := ADR(SendTelegram),
					mSendDataLen := WritePointer);

// Forward to mirror channel
M_MirrorData(Data := ADR(SendTelegram), DataLen := WritePointer);
END_METHOD

METHOD PROTECTED M_ProcessRAC : BOOL
(**************************************************************************************
 * 	Application		:	BoxControl Framework
 *	Revision		:	$Revision: 404529 $
 *	Revision date	:	$Date: 2018-04-23 08:21:38 +0200 (Mo., 23 Apr 2018) $
 *	Last changed by	:	$Author: b7bolm $
 *	URL				:	$URL: http://almscdc.swisslog.com/repo/SWPD/Development/BoxControlFramework/20_Release/trunk/01_Software/BCF/BCF/JumpStart/20_Product/10_App/11_Com/10_Lib/10_Conv/12_MFCS/11_SIS/FB_SIS_MsgManager_6_1.TcPOU $
 *
 *	Purpose			:	Send RAC Robot Task Complete
 *
 * ------------------------------------------------------------------------------------
 *	Copyright Swisslog [IP AG], Switzerland. All rights reserved.
 * 
 * ------------------------------------------------------------------------------------
 *	
 * 	Revision History: 
 *
 * 	VERSION			DATE			INITIALS			DESCRIPTION
 *	0.1				01.01.2001		swl					Example
 *
 *************************************************************************************)
VAR_INPUT
	meChannelSrc				: E_MFCS_Channel; // Source communicaton channel	
	mpRAC						: POINTER TO ST_ITC_RAC;
END_VAR
(**************************************************************************************************************
 	Check if a telegram needs to be send
***************************************************************************************************************)
// If settings allow sending a RAC 	
IF  Settings.Telegrams.SendRAC THEN
	// If the source of the request is this channel or is undefined
	IF meChannelSrc = Settings.MFCS_Channel OR
		meChannelSrc = E_MFCS_Channel.BEGIN_CHANNEL THEN
		;//Proceed
	ELSE // Source is a different MFCS Connection
		// Dont send a telegram		
		RETURN;
	END_IF	
ELSE
	// Dont send a telegram		
	RETURN;
END_IF

(**************************************************************************************************************
 	ITC - Map generic data to type
***************************************************************************************************************)
MEMCPY(destAddr := ADR(RAC_ITC), srcAddr := mpRAC, n := SIZEOF(RAC_ITC));

(**************************************************************************************************************
 	Formatting data
***************************************************************************************************************)
// Get position
RAC.Position := F_StuffString(
					InputString 	:= RAC_ITC.Position, 
					StringLength	:= SIS_6_1.POSITION_STRINGLENGTH, 
					StuffCharacter 	:= '0',
					LeftAligned		:= FALSE);

// Get command data index 
RAC.CommandDataIndex := F_StuffString(
				InputString 	:= DINT_TO_STRING(RAC_ITC.CommandDataIndex), 
				StringLength	:= SIS_6_1.RAC_COMMAND_DATA_INDEX_STRINGLENGTH, 
				StuffCharacter 	:= '0',
				LeftAligned		:= FALSE);
					
// Get assignment ID 
RAC.AssignmentID := F_StuffString(
						InputString 	:= UDINT_TO_STRING(RAC_ITC.AssignmentID), 
						StringLength	:= SIS_6_1.ASSIGNMENT_ID_STRINGLENGTH, 
						StuffCharacter 	:= '0',
						LeftAligned		:= FALSE);

// Get group ID 
RAC.GroupID := 	F_StuffString(
					InputString 	:= ULINT_TO_STRING(RAC_ITC.GroupID), 
					StringLength	:= SIS_6_1.GROUP_ID_STRINGLENGTH, 
					StuffCharacter 	:= '0',
					LeftAligned		:= FALSE);

// Get return code 
RAC.ReturnCode := F_StuffString(
					InputString 	:= INT_TO_STRING(RAC_ITC.eReturnCode), 
					StringLength	:= SIS_6_1.ERRORCODE_STRINGLENGTH, 
					StuffCharacter 	:= '0',
					LeftAligned		:= FALSE);

(**************************************************************************************************************
 	Build string and add to Base Driver
***************************************************************************************************************)
MEMSET(destAddr := ADR(SendTelegram), 0, SIZEOF(SendTelegram));
WritePointer := 0;

F_AssembleByteStream(
	pSrc:= ADR('RAC'), 
	SrcLen:= 3, 
	pDest:= ADR(SendTelegram), 
	DestLen:= SIZEOF(SendTelegram), 
	WritePointer:= WritePointer);
	
F_AssembleByteStream(
	pSrc:= ADR(RAC.Position), 
	SrcLen:= INT_TO_UDINT(LEN(RAC.Position)), 
	pDest:= ADR(SendTelegram), 
	DestLen:= SIZEOF(SendTelegram), 
	WritePointer:= WritePointer);

F_AssembleByteStream(
	pSrc:= ADR(RAC.CommandDataIndex), 
	SrcLen:= INT_TO_UDINT(LEN(RAC.CommandDataIndex)), 
	pDest:= ADR(SendTelegram), 
	DestLen:= SIZEOF(SendTelegram), 
	WritePointer:= WritePointer);

F_AssembleByteStream(
	pSrc:= ADR(RAC.AssignmentID), 
	SrcLen:= INT_TO_UDINT(LEN(RAC.AssignmentID)), 
	pDest:= ADR(SendTelegram), 
	DestLen:= SIZEOF(SendTelegram), 
	WritePointer:= WritePointer);

F_AssembleByteStream(
	pSrc:= ADR(RAC.GroupID), 
	SrcLen:= INT_TO_UDINT(LEN(RAC.GroupID)), 
	pDest:= ADR(SendTelegram), 
	DestLen:= SIZEOF(SendTelegram), 
	WritePointer:= WritePointer);

F_AssembleByteStream(
	pSrc:= ADR(RAC.ReturnCode), 
	SrcLen:= INT_TO_UDINT(LEN(RAC.ReturnCode)), 
	pDest:= ADR(SendTelegram), 
	DestLen:= SIZEOF(SendTelegram), 
	WritePointer:= WritePointer);

// Add to buffer of Base Driver
M_ProcessRAC := fbBaseDriver.M_SendAppData(
					mpSendData := ADR(SendTelegram),
					mSendDataLen := WritePointer);

// Forward to mirror channel
M_MirrorData(Data := ADR(SendTelegram), DataLen := WritePointer);
END_METHOD

METHOD PROTECTED M_ProcessRAQ : BOOL
(**************************************************************************************
 * 	Application		:	BoxControl Framework
 *	Revision		:	$Revision: 404529 $
 *	Revision date	:	$Date: 2018-04-23 08:21:38 +0200 (Mo., 23 Apr 2018) $
 *	Last changed by	:	$Author: b7bolm $
 *	URL				:	$URL: http://almscdc.swisslog.com/repo/SWPD/Development/BoxControlFramework/20_Release/trunk/01_Software/BCF/BCF/JumpStart/20_Product/10_App/11_Com/10_Lib/10_Conv/12_MFCS/11_SIS/FB_SIS_MsgManager_6_1.TcPOU $
 *
 *	Purpose			:	Send RAQ
 *
 * ------------------------------------------------------------------------------------
 *	Copyright Swisslog [IP AG], Switzerland. All rights reserved.
 * 
 * ------------------------------------------------------------------------------------
 *	
 * 	Revision History: 
 *
 * 	VERSION			DATE			INITIALS			DESCRIPTION
 *	0.1				01.01.2001		swl					Example
 *
 **************************************************************************************)
VAR_INPUT
 	meChannelSrc		: E_MFCS_Channel; // Source communicaton channel
	mpRAQ				: POINTER TO ST_ITC_RAQ; // Pointer to RAQ
END_VAR
(**************************************************************************************************************
 	Check if a telegram needs to be send
***************************************************************************************************************)
// If settings allow sending a RAQ 	
IF  Settings.Telegrams.SendRAQ THEN
	// If the source of the request is this channel or is undefined
	IF meChannelSrc = Settings.MFCS_Channel OR
		meChannelSrc = E_MFCS_Channel.BEGIN_CHANNEL THEN
		;//Proceed
	ELSE // Source is a different MFCS Connection
		// Dont send a telegram		
		RETURN;
	END_IF	
ELSE
	// Dont send a telegram		
	RETURN;
END_IF

(**************************************************************************************************************
 	ITC - Map generic data to type
***************************************************************************************************************)
MEMCPY(destAddr := ADR(RAQ_ITC), srcAddr := mpRAQ, n := SIZEOF(RAQ_ITC));

(**************************************************************************************************************
 	Formatting data
***************************************************************************************************************)
// Get position
RAQ.Position	:= 	F_StuffString(
						InputString 	:= RAQ_ITC.Position, 
						StringLength	:= SIS_6_1.POSITION_STRINGLENGTH, 
						StuffCharacter 	:= '0',
						LeftAligned		:= FALSE);

// Get group ID
RAQ.GroupID := F_StuffString(
				InputString		:= ULINT_TO_STRING(RAQ_ITC.GroupID),
				StringLength	:= SIS_6_1.GROUP_ID_STRINGLENGTH,
				StuffCharacter	:= '0',
				LeftAligned		:= FALSE);

// Get number of RA
RAQ.NumberOfRA := F_StuffString(
				InputString		:= INT_TO_STRING(RAQ_ITC.NumberOfRA),
				StringLength	:= SIS_6_1.RAQ_NUMBER_OF_RA_STRINGLENGTH,
				StuffCharacter	:= '0',
				LeftAligned		:= FALSE);
					
(**************************************************************************************************************
 	Build string and add to Base Driver
***************************************************************************************************************)
MEMSET(destAddr := ADR(SendTelegram), 0, SIZEOF(SendTelegram));
WritePointer := 0;

F_AssembleByteStream(
	pSrc:= ADR('RAQ'), 
	SrcLen:= 3, 
	pDest:= ADR(SendTelegram), 
	DestLen:= SIZEOF(SendTelegram), 
	WritePointer:= WritePointer);
	
F_AssembleByteStream(
	pSrc:= ADR(RAQ.Position), 
	SrcLen:= INT_TO_UDINT(LEN(RAQ.Position)), 
	pDest:= ADR(SendTelegram), 
	DestLen:= SIZEOF(SendTelegram), 
	WritePointer:= WritePointer);

F_AssembleByteStream(
	pSrc:= ADR(RAQ.GroupID), 
	SrcLen:= INT_TO_UDINT(LEN(RAQ.GroupID)), 
	pDest:= ADR(SendTelegram), 
	DestLen:= SIZEOF(SendTelegram), 
	WritePointer:= WritePointer);

F_AssembleByteStream(
	pSrc:= ADR(RAQ.NumberOfRA), 
	SrcLen:= INT_TO_UDINT(LEN(RAQ.NumberOfRA)), 
	pDest:= ADR(SendTelegram), 
	DestLen:= SIZEOF(SendTelegram), 
	WritePointer:= WritePointer);	
	
// Add to buffer of Base Driver
M_ProcessRAQ := fbBaseDriver.M_SendAppData(
					mpSendData := ADR(SendTelegram),
					mSendDataLen := WritePointer);

// Forward to mirror channel
M_MirrorData(Data := ADR(SendTelegram), DataLen := WritePointer);
END_METHOD

METHOD PROTECTED M_ProcessRDR : BOOL
(**************************************************************************************
 * 	Application		:	BoxControl Framework
 *	Revision		:	$Revision: 404529 $
 *	Revision date	:	$Date: 2018-04-23 08:21:38 +0200 (Mo., 23 Apr 2018) $
 *	Last changed by	:	$Author: b7bolm $
 *	URL				:	$URL: http://almscdc.swisslog.com/repo/SWPD/Development/BoxControlFramework/20_Release/trunk/01_Software/BCF/BCF/JumpStart/20_Product/10_App/11_Com/10_Lib/10_Conv/12_MFCS/11_SIS/FB_SIS_MsgManager_6_1.TcPOU $
 *
 *	Purpose			:	Send RDR
 *
 * ------------------------------------------------------------------------------------
 *	Copyright Swisslog [IP AG], Switzerland. All rights reserved.
 * 
 * ------------------------------------------------------------------------------------
 *	
 * 	Revision History: 
 *
 * 	VERSION			DATE			INITIALS			DESCRIPTION
 *	0.1				04.01.2016		Kay Röder			Initial programming
 *
 **************************************************************************************)
VAR_INPUT
	meChannelSrc		: E_MFCS_Channel; // Source communicaton channel
	mpRDR				: POINTER TO ST_ITC_RDR; // Pointer to RDR
END_VAR
(**************************************************************************************************************
 	Check if a telegram needs to be send
***************************************************************************************************************)
// If settings allow sending a RDR 	
IF  Settings.Telegrams.SendRDR THEN
	// If the source of the request is this channel or is undefined
	IF meChannelSrc = Settings.MFCS_Channel OR
		meChannelSrc = E_MFCS_Channel.BEGIN_CHANNEL THEN
		;//Proceed
	ELSE // Source is a different MFCS Connection
		// Dont send a telegram		
		RETURN;
	END_IF	
ELSE
	// Dont send a telegram		
	RETURN;
END_IF

(**************************************************************************************************************
 	ITC - Map generic data to type
***************************************************************************************************************)
MEMCPY(destAddr := ADR(RDR_ITC), srcAddr := mpRDR, n := SIZEOF(RDR_ITC));

(**************************************************************************************************************
 	Formatting data
***************************************************************************************************************)
// Get position
RDR.Position := F_StuffString(
					InputString		:= RDR_ITC.Position,
					StringLength	:= SIS_6_1.POSITION_STRINGLENGTH,
					StuffCharacter	:= '0',
					LeftAligned		:= FALSE);

// Get command data index
RDR.CommandDataIndex := F_StuffString(
						InputString		:= DINT_TO_STRING(RDR_ITC.CommandDataIndex),
						StringLength	:= SIS_6_1.RDR_COMMAND_DATA_INDEX_STRINGLENGTH,
						StuffCharacter	:= '0',
						LeftAligned		:= FALSE);
						
// Get assignment ID
RDR.AssignmentID := F_StuffString(
						InputString		:= UDINT_TO_STRING(RDR_ITC.AssignmentID),
						StringLength	:= SIS_6_1.ASSIGNMENT_ID_STRINGLENGTH,
						StuffCharacter	:= '0',
						LeftAligned		:= FALSE);
						
// Get group ID
RDR.GroupID := F_StuffString(
				InputString		:= ULINT_TO_STRING(RDR_ITC.GroupID),
				StringLength	:= SIS_6_1.GROUP_ID_STRINGLENGTH,
				StuffCharacter	:= '0',
				LeftAligned		:= FALSE);

// Get return code
RDR.ReturnCode := F_StuffString(
						InputString		:= INT_TO_STRING(RDR_ITC.ReturnCode),
						StringLength	:= SIS_6_1.ERRORCODE_STRINGLENGTH,
						StuffCharacter	:= '0',
						LeftAligned		:= FALSE);
						
(**************************************************************************************************************
 	Build string and add to Base Driver
***************************************************************************************************************)
MEMSET(destAddr := ADR(SendTelegram), 0, SIZEOF(SendTelegram));
WritePointer := 0;

F_AssembleByteStream(
	pSrc:= ADR('RDR'), 
	SrcLen:= 3, 
	pDest:= ADR(SendTelegram), 
	DestLen:= SIZEOF(SendTelegram), 
	WritePointer:= WritePointer);
	
F_AssembleByteStream(
	pSrc:= ADR(RDR.Position), 
	SrcLen:= INT_TO_UDINT(LEN(RDR.Position)), 
	pDest:= ADR(SendTelegram), 
	DestLen:= SIZEOF(SendTelegram), 
	WritePointer:= WritePointer);
	
F_AssembleByteStream(
	pSrc:= ADR(RDR.CommandDataIndex), 
	SrcLen:= INT_TO_UDINT(LEN(RDR.CommandDataIndex)), 
	pDest:= ADR(SendTelegram), 
	DestLen:= SIZEOF(SendTelegram), 
	WritePointer:= WritePointer);
	
F_AssembleByteStream(
	pSrc:= ADR(RDR.AssignmentID), 
	SrcLen:= INT_TO_UDINT(LEN(RDR.AssignmentID)), 
	pDest:= ADR(SendTelegram), 
	DestLen:= SIZEOF(SendTelegram), 
	WritePointer:= WritePointer);
	
F_AssembleByteStream(
	pSrc:= ADR(RDR.GroupID), 
	SrcLen:= INT_TO_UDINT(LEN(RDR.GroupID)), 
	pDest:= ADR(SendTelegram), 
	DestLen:= SIZEOF(SendTelegram), 
	WritePointer:= WritePointer);

F_AssembleByteStream(
	pSrc:= ADR(RDR.ReturnCode), 
	SrcLen:= INT_TO_UDINT(LEN(RDR.ReturnCode)), 
	pDest:= ADR(SendTelegram), 
	DestLen:= SIZEOF(SendTelegram), 
	WritePointer:= WritePointer);

// Add to buffer of Base Driver
M_ProcessRDR := fbBaseDriver.M_SendAppData(
					mpSendData := ADR(SendTelegram),
					mSendDataLen := WritePointer);

// Forward to mirror channel
M_MirrorData(Data := ADR(SendTelegram), DataLen := WritePointer);
END_METHOD

METHOD PROTECTED M_ProcessRTR : BOOL
(**************************************************************************************
 * 	Application		:	BoxControl Framework
 *	Revision		:	$Revision: 404529 $
 *	Revision date	:	$Date: 2018-04-23 08:21:38 +0200 (Mo., 23 Apr 2018) $
 *	Last changed by	:	$Author: b7bolm $
 *	URL				:	$URL: http://almscdc.swisslog.com/repo/SWPD/Development/BoxControlFramework/20_Release/trunk/01_Software/BCF/BCF/JumpStart/20_Product/10_App/11_Com/10_Lib/10_Conv/12_MFCS/11_SIS/FB_SIS_MsgManager_6_1.TcPOU $
 *
 *	Purpose			:	Send RTR
 *
 * ------------------------------------------------------------------------------------
 *	Copyright Swisslog [IP AG], Switzerland. All rights reserved.
 * 
 * ------------------------------------------------------------------------------------
 *	
 * 	Revision History: 
 *
 * 	VERSION			DATE			INITIALS			DESCRIPTION
 *	0.1				01.01.2001		swl					Example
 *
 **************************************************************************************)
VAR_INPUT
 	meChannelSrc		: E_MFCS_Channel; // Source communicaton channel
	mpRTR				: POINTER TO ST_ITC_RTR; // Pointer to RTR
END_VAR
(**************************************************************************************************************
 	Check if a telegram needs to be send
***************************************************************************************************************)
// If settings allow sending a RTR 	
IF  Settings.Telegrams.SendRTR THEN
	// If the source of the request is this channel or is undefined
	IF meChannelSrc = Settings.MFCS_Channel OR
		meChannelSrc = E_MFCS_Channel.BEGIN_CHANNEL THEN
		;//Proceed
	ELSE // Source is a different MFCS Connection
		// Dont send a telegram		
		RETURN;
	END_IF	
ELSE
	// Dont send a telegram		
	RETURN;
END_IF

(**************************************************************************************************************
 	ITC - Map generic data to type
***************************************************************************************************************)
MEMCPY(destAddr := ADR(RTR_ITC), srcAddr := mpRTR, n := SIZEOF(RTR_ITC));

(**************************************************************************************************************
 	Formatting data
***************************************************************************************************************)
// Get position
RTR.Position	:= 	F_StuffString(
						InputString 	:= RTR_ITC.Position, 
						StringLength	:= SIS_6_1.POSITION_STRINGLENGTH, 
						StuffCharacter 	:= '0',
						LeftAligned		:= FALSE);

// Get error code 
RTR.ReturnCode := F_StuffString(
					InputString 	:= INT_TO_STRING(RTR_ITC.ReturnCode), 
					StringLength	:= SIS_6_1.ERRORCODE_STRINGLENGTH, 
					StuffCharacter 	:= '0',
					LeftAligned		:= FALSE);
					
(**************************************************************************************************************
 	Build string and add to Base Driver
***************************************************************************************************************)
MEMSET(destAddr := ADR(SendTelegram), 0, SIZEOF(SendTelegram));
WritePointer := 0;

F_AssembleByteStream(
	pSrc:= ADR('RTR'), 
	SrcLen:= 3, 
	pDest:= ADR(SendTelegram), 
	DestLen:= SIZEOF(SendTelegram), 
	WritePointer:= WritePointer);
	
F_AssembleByteStream(
	pSrc:= ADR(RTR.Position), 
	SrcLen:= INT_TO_UDINT(LEN(RTR.Position)), 
	pDest:= ADR(SendTelegram), 
	DestLen:= SIZEOF(SendTelegram), 
	WritePointer:= WritePointer);

F_AssembleByteStream(
	pSrc:= ADR(RTR.ReturnCode), 
	SrcLen:= INT_TO_UDINT(LEN(RTR.ReturnCode)), 
	pDest:= ADR(SendTelegram), 
	DestLen:= SIZEOF(SendTelegram), 
	WritePointer:= WritePointer);

// Add to buffer of Base Driver
M_ProcessRTR := fbBaseDriver.M_SendAppData(
					mpSendData := ADR(SendTelegram),
					mSendDataLen := WritePointer);

// Forward to mirror channel
M_MirrorData(Data := ADR(SendTelegram), DataLen := WritePointer);
END_METHOD

METHOD PROTECTED M_ProcessSCR : BOOL
(**************************************************************************************
 * 	Application		:	BoxControl Framework
 *	Revision		:	$Revision: 404529 $
 *	Revision date	:	$Date: 2018-04-23 08:21:38 +0200 (Mo., 23 Apr 2018) $
 *	Last changed by	:	$Author: b7bolm $
 *	URL				:	$URL: http://almscdc.swisslog.com/repo/SWPD/Development/BoxControlFramework/20_Release/trunk/01_Software/BCF/BCF/JumpStart/20_Product/10_App/11_Com/10_Lib/10_Conv/12_MFCS/11_SIS/FB_SIS_MsgManager_6_1.TcPOU $
 *
 *	Purpose			:	Send SCR.
 *
 * ------------------------------------------------------------------------------------
 *	Copyright Swisslog [IP AG], Switzerland. All rights reserved.
 * 
 * ------------------------------------------------------------------------------------
 *	
 * 	Revision History: 
 *
 * 	VERSION			DATE			INITIALS			DESCRIPTION
 *	0.1				01.01.2001		swl					Example
 *
 **************************************************************************************)
VAR_INPUT
 	meChannelSrc		: E_MFCS_Channel; // Source communicaton channel
	mpSCR				: POINTER TO ST_ITC_SCR; // Pointer to SCR
END_VAR
(**************************************************************************************************************
 	Check if a telegram needs to be send
***************************************************************************************************************)
// If settings allow sending a SCR 	
IF  Settings.Telegrams.SendSCR THEN
	// If the source of the request is this channel or is undefined
	IF meChannelSrc = Settings.MFCS_Channel OR
		meChannelSrc = E_MFCS_Channel.BEGIN_CHANNEL THEN
		;//Proceed
	ELSE // Source is a different MFCS Connection
		// Dont send a telegram		
		RETURN;
	END_IF	
ELSE
	// Dont send a telegram		
	RETURN;
END_IF

(**************************************************************************************************************
 	ITC - Map generic data to type
***************************************************************************************************************)
MEMCPY(destAddr := ADR(SCR_ITC), srcAddr := mpSCR, n := SIZEOF(SCR_ITC));

(**************************************************************************************************************
 	Formatting data
***************************************************************************************************************)

// Get Subsystem name 
SCR.SubsystemName := F_StuffString(
							InputString 	:= SCR_ITC.SubsystemName, 
							StringLength	:= SIS_6_1.POSITION_STRINGLENGTH, 
							StuffCharacter 	:= '0',
							LeftAligned		:= FALSE);

// Get Code 
SCR.Code := F_StuffString(
				InputString 	:= INT_TO_STRING(SCR_ITC.Code), 
				StringLength	:= SIS_6_1.CONTROLCODE_STRINGLENGTH, 
				StuffCharacter 	:= '0',
				LeftAligned		:= FALSE);

// Get Variable 
SCR.Variable := F_StuffString(
					InputString 	:= DINT_TO_STRING(SCR_ITC.Variable), 
					StringLength	:= SIS_6_1.CONTROLVARIABLE_STRINGLENGTH, 
					StuffCharacter 	:= '0',
					LeftAligned		:= FALSE);

// Get ErrorCode
SCR.ReturnCode := F_StuffString(
						InputString 	:= INT_TO_STRING(SCR_ITC.ReturnCode), 
						StringLength	:= SIS_6_1.ERRORCODE_STRINGLENGTH, 
						StuffCharacter 	:= '0',
						LeftAligned		:= FALSE);


(**************************************************************************************************************
 	Build string and add to Base Driver
***************************************************************************************************************)
MEMSET(destAddr := ADR(SendTelegram), 0, SIZEOF(SendTelegram));
WritePointer := 0;

F_AssembleByteStream(
	pSrc:= ADR('SCR'), 
	SrcLen:= 3, 
	pDest:= ADR(SendTelegram), 
	DestLen:= SIZEOF(SendTelegram), 
	WritePointer:= WritePointer);
	
F_AssembleByteStream(
	pSrc:= ADR(SCR.SubsystemName), 
	SrcLen:= INT_TO_UDINT(LEN(SCR.SubsystemName)), 
	pDest:= ADR(SendTelegram), 
	DestLen:= SIZEOF(SendTelegram), 
	WritePointer:= WritePointer);

F_AssembleByteStream(
	pSrc:= ADR(SCR.Code), 
	SrcLen:= INT_TO_UDINT(LEN(SCR.Code)), 
	pDest:= ADR(SendTelegram), 
	DestLen:= SIZEOF(SendTelegram), 
	WritePointer:= WritePointer);

F_AssembleByteStream(
	pSrc:= ADR(SCR.Variable), 
	SrcLen:= INT_TO_UDINT(LEN(SCR.Variable)), 
	pDest:= ADR(SendTelegram), 
	DestLen:= SIZEOF(SendTelegram), 
	WritePointer:= WritePointer);

F_AssembleByteStream(
	pSrc:= ADR(SCR.ReturnCode), 
	SrcLen:= INT_TO_UDINT(LEN(SCR.ReturnCode)), 
	pDest:= ADR(SendTelegram), 
	DestLen:= SIZEOF(SendTelegram), 
	WritePointer:= WritePointer);


// Add to buffer of Base Driver
M_ProcessSCR := fbBaseDriver.M_SendAppData(
					mpSendData := ADR(SendTelegram),
					mSendDataLen := WritePointer);

// Forward to mirror channel
M_MirrorData(Data := ADR(SendTelegram), DataLen := WritePointer);
END_METHOD

METHOD PROTECTED M_ProcessSDI : BOOL
(**************************************************************************************
 * 	Application		:	BoxControl Framework
 *	Revision		:	$Revision: 404529 $
 *	Revision date	:	$Date: 2018-04-23 08:21:38 +0200 (Mo., 23 Apr 2018) $
 *	Last changed by	:	$Author: b7bolm $
 *	URL				:	$URL: http://almscdc.swisslog.com/repo/SWPD/Development/BoxControlFramework/20_Release/trunk/01_Software/BCF/BCF/JumpStart/20_Product/10_App/11_Com/10_Lib/10_Conv/12_MFCS/11_SIS/FB_SIS_MsgManager_6_1.TcPOU $
 *
 *	Purpose			:	Send SDI
 *
 * ------------------------------------------------------------------------------------
 *	Copyright Swisslog [IP AG], Switzerland. All rights reserved.
 * 
 * ------------------------------------------------------------------------------------
 *	
 * 	Revision History: 
 *
 * 	VERSION			DATE			INITIALS			DESCRIPTION
 *	0.1				01.01.2001		swl					Example
 *
 **************************************************************************************)
VAR_INPUT
 	meChannelSrc		: E_MFCS_Channel; // Source communicaton channel
	mpSDI				: POINTER TO ST_ITC_SDI; // Pointer to SDI
END_VAR
(**************************************************************************************************************
 	Check if a telegram needs to be send
***************************************************************************************************************)
// If settings allow sending a SDI 	
IF  Settings.Telegrams.SendSDI THEN
	// If the source of the request is this channel or is undefined
	IF meChannelSrc = Settings.MFCS_Channel OR
		meChannelSrc = E_MFCS_Channel.BEGIN_CHANNEL THEN
		;//Proceed
	ELSE // Source is a different MFCS Connection
		// Dont send a telegram		
		RETURN;
	END_IF	
ELSE
	// Dont send a telegram		
	RETURN;
END_IF


(**************************************************************************************************************
 	ITC - Map generic data to type
***************************************************************************************************************)
MEMCPY(destAddr := ADR(SDI_ITC), srcAddr := mpSDI, n := SIZEOF(SDI_ITC));

(**************************************************************************************************************
 	Formatting data
***************************************************************************************************************)

// Get SignalNumber 
SDI.SignalNumber := F_StuffString(
						InputString 	:= INT_TO_STRING(SDI_ITC.SignalNumber), 
						StringLength	:= SIS_6_1.SDI_SIGNALNUMBER_STRINGLENGTH, 
						StuffCharacter 	:= '0',
						LeftAligned		:= FALSE);

// Get SignalState 
SDI.SignalState := INT_TO_STRING(BOOL_TO_INT(SDI_ITC.SignalState));

// Get Error Code 
SDI.ReturnCode := F_StuffString(
					InputString 	:= INT_TO_STRING(SDI_ITC.ReturnCode), 
					StringLength	:= SIS_6_1.ERRORCODE_STRINGLENGTH, 
					StuffCharacter 	:= '0',
					LeftAligned		:= FALSE);

(**************************************************************************************************************
 	Build string and add to Base Driver
***************************************************************************************************************)
MEMSET(destAddr := ADR(SendTelegram), 0, SIZEOF(SendTelegram));
WritePointer := 0;

F_AssembleByteStream(
	pSrc:= ADR('SDI'), 
	SrcLen:= 3, 
	pDest:= ADR(SendTelegram), 
	DestLen:= SIZEOF(SendTelegram), 
	WritePointer:= WritePointer);
	
F_AssembleByteStream(
	pSrc:= ADR(SDI.SignalNumber), 
	SrcLen:= INT_TO_UDINT(LEN(SDI.SignalNumber)), 
	pDest:= ADR(SendTelegram), 
	DestLen:= SIZEOF(SendTelegram), 
	WritePointer:= WritePointer);
	
F_AssembleByteStream(
	pSrc:= ADR(SDI.SignalState), 
	SrcLen:= INT_TO_UDINT(LEN(SDI.SignalState)), 
	pDest:= ADR(SendTelegram), 
	DestLen:= SIZEOF(SendTelegram), 
	WritePointer:= WritePointer);	
	
F_AssembleByteStream(
	pSrc:= ADR(SDI.ReturnCode), 
	SrcLen:= INT_TO_UDINT(LEN(SDI.ReturnCode)), 
	pDest:= ADR(SendTelegram), 
	DestLen:= SIZEOF(SendTelegram), 
	WritePointer:= WritePointer);

// Add to buffer of Base Driver
M_ProcessSDI := fbBaseDriver.M_SendAppData(
					mpSendData := ADR(SendTelegram),
					mSendDataLen := WritePointer);

// Forward to mirror channel
M_MirrorData(Data := ADR(SendTelegram), DataLen := WritePointer);
END_METHOD

METHOD PROTECTED M_ProcessSIR : BOOL
(**************************************************************************************
 * 	Application		:	BoxControl Framework
 *	Revision		:	$Revision: 404529 $
 *	Revision date	:	$Date: 2018-04-23 08:21:38 +0200 (Mo., 23 Apr 2018) $
 *	Last changed by	:	$Author: b7bolm $
 *	URL				:	$URL: http://almscdc.swisslog.com/repo/SWPD/Development/BoxControlFramework/20_Release/trunk/01_Software/BCF/BCF/JumpStart/20_Product/10_App/11_Com/10_Lib/10_Conv/12_MFCS/11_SIS/FB_SIS_MsgManager_6_1.TcPOU $
 *
 *	Purpose			:	Send SIR
 *
 * ------------------------------------------------------------------------------------
 *	Copyright Swisslog [IP AG], Switzerland. All rights reserved.
 * 
 * ------------------------------------------------------------------------------------
 *	
 * 	Revision History: 
 *
 * 	VERSION			DATE			INITIALS			DESCRIPTION
 *	0.1				01.01.2001		swl					Example
 *
 **************************************************************************************)
VAR_INPUT
 	meChannelSrc		: E_MFCS_Channel; // Source communicaton channel
	mpSIR				: POINTER TO ST_ITC_SIR; // Pointer to SIR
END_VAR
(**************************************************************************************************************
 	Check if a telegram needs to be send
***************************************************************************************************************)
// If settings allow sending a SIR 	
IF  Settings.Telegrams.SendSIR THEN
	// If the source of the request is this channel or is undefined
	IF meChannelSrc = Settings.MFCS_Channel OR
		meChannelSrc = E_MFCS_Channel.BEGIN_CHANNEL THEN
		;//Proceed
	ELSE // Source is a different MFCS Connection
		// Dont send a telegram		
		RETURN;
	END_IF	
ELSE
	// Dont send a telegram		
	RETURN;
END_IF

(**************************************************************************************************************
 	ITC - Map generic data to type
***************************************************************************************************************)
MEMCPY(destAddr := ADR(SIR_ITC), srcAddr := mpSIR, n := SIZEOF(SIR_ITC));

(**************************************************************************************************************
 	Formatting data
***************************************************************************************************************)

// Get SIS-Number 
SIR.Position := F_StuffString(
							InputString 	:= SIR_ITC.Position, 
							StringLength	:= SIS_6_1.POSITION_STRINGLENGTH, 
							StuffCharacter 	:= '0',
							LeftAligned		:= FALSE);
							
// Get Code 
SIR.Code := F_StuffString(
				InputString 	:= INT_TO_STRING(SIR_ITC.Code), 
				StringLength	:= SIS_6_1.SIR_CODE_STRINGLENGTH, 
				StuffCharacter 	:= '0',
				LeftAligned		:= FALSE);

// Get TU-ID 
SIR.TU_ID := F_StuffString(
				InputString 	:= SIR_ITC.TU_ID, 
				StringLength	:= SIS_6_1.TU_ID_STRINGLENGTH, 
				StuffCharacter 	:= ' ',
				LeftAligned		:= FALSE);

// Get counter value
SIR.Counter1 := F_StuffString(
					InputString 	:= DINT_TO_STRING(SIR_ITC.Counter1), 
					StringLength	:= SIS_6_1.SIR_COUNTER_STRINGLENGTH, 
					StuffCharacter 	:= '0',
					LeftAligned		:= FALSE);

// Get counter value
SIR.Counter2 := F_StuffString(
					InputString 	:= DINT_TO_STRING(SIR_ITC.Counter2), 
					StringLength	:= SIS_6_1.SIR_COUNTER_STRINGLENGTH, 
					StuffCharacter 	:= '0',
					LeftAligned		:= FALSE);

// Get counter value
SIR.Counter3 := F_StuffString(
					InputString 	:= DINT_TO_STRING(SIR_ITC.Counter3), 
					StringLength	:= SIS_6_1.SIR_COUNTER_STRINGLENGTH, 
					StuffCharacter 	:= '0',
					LeftAligned		:= FALSE);

// Get counter value
SIR.Counter4 := F_StuffString(
					InputString 	:= DINT_TO_STRING(SIR_ITC.Counter4), 
					StringLength	:= SIS_6_1.SIR_COUNTER_STRINGLENGTH, 
					StuffCharacter 	:= '0',
					LeftAligned		:= FALSE);
		
// Get counter value		
SIR.Counter5 := F_StuffString(
					InputString 	:= DINT_TO_STRING(SIR_ITC.Counter5), 
					StringLength	:= SIS_6_1.SIR_COUNTER_STRINGLENGTH, 
					StuffCharacter 	:= '0',
					LeftAligned		:= FALSE);
		
// Get error code
SIR.ReturnCode := F_StuffString(
					InputString 	:= INT_TO_STRING(SIR_ITC.eReturnCode), 
					StringLength	:= SIS_6_1.ERRORCODE_STRINGLENGTH, 
					StuffCharacter 	:= '0',
					LeftAligned		:= FALSE);


(**************************************************************************************************************
 	Build string and add to Base Driver
***************************************************************************************************************)
MEMSET(destAddr := ADR(SendTelegram), 0, SIZEOF(SendTelegram));
WritePointer := 0;

F_AssembleByteStream(
	pSrc:= ADR('SIR'), 
	SrcLen:= 3, 
	pDest:= ADR(SendTelegram), 
	DestLen:= SIZEOF(SendTelegram), 
	WritePointer:= WritePointer);
	
F_AssembleByteStream(
	pSrc:= ADR(SIR.Position), 
	SrcLen:= INT_TO_UDINT(LEN(SIR.Position)), 
	pDest:= ADR(SendTelegram), 
	DestLen:= SIZEOF(SendTelegram), 
	WritePointer:= WritePointer);
	
